SPLINE
SPL {X  -165.650, Y  +492.090, Z    +0.000, E1   -45.292, E3 +369321.420}
SPL {X  -165.650, Y  +498.857, Z    +0.000, E1   -45.339, E3 +369334.757}
SPL {X  -165.650, Y  +505.115, Z    +0.000, E1   -45.299, E3 +369347.706}
SPL {X  -165.650, Y  +510.931, Z    +0.000, E1   -45.250, E3 +369359.696}
SPL {X  -165.650, Y  +516.157, Z    +0.000, E1   -45.240, E3 +369370.371}
SPL {X  -165.650, Y  +521.049, Z    +0.000, E1   -45.236, E3 +369380.323}
SPL {X  -165.650, Y  +527.050, Z    +0.000, E1   -45.345, E3 +369391.820}
SPL {X  -165.650, Y  +532.042, Z    +0.000, E1   -45.233, E3 +369402.563}
SPL {X  -165.650, Y  +537.290, Z    +0.000, E1   -45.204, E3 +369413.404}
SPL {X  -165.650, Y  +544.196, Z    +0.000, E1   -45.432, E3 +369426.078}
SPL {X  -165.650, Y  +548.678, Z    +0.000, E1   -45.162, E3 +369436.642}
SPL {X  -165.650, Y  +554.600, Z    +0.000, E1   -45.345, E3 +369447.619}
SPL {X  -165.650, Y  +559.896, Z    +0.000, E1   -45.150, E3 +369459.474}
SPL {X  -165.650, Y  +566.830, Z    +0.000, E1   -45.346, E3 +369472.454}
SPL {X  -165.650, Y  +573.074, Z    +0.000, E1   -45.379, E3 +369484.785}
SPL {X  -165.650, Y  +579.360, Z    +0.000, E1   -45.300, E3 +369498.070}
SPL {X  -165.650, Y  +584.577, Z    +0.000, E1   -45.167, E3 +369509.293}
SPL {X  -165.650, Y  +590.060, Z    +0.000, E1   -45.221, E3 +369520.184}
SPL {X  -165.650, Y  +596.611, Z    +0.000, E1   -45.390, E3 +369532.421}
SPL {X  -165.650, Y  +603.637, Z    +0.000, E1   -45.296, E3 +369547.339}
SPL {X  -165.650, Y  +610.850, Z    +0.000, E1   -45.208, E3 +369562.348}
SPL {X  -165.650, Y  +617.450, Z    +0.000, E1   -45.402, E3 +369574.550}
SPL {X  -165.650, Y  +622.720, Z    +0.000, E1   -45.272, E3 +369585.948}
SPL {X  -165.650, Y  +627.828, Z    +0.000, E1   -45.174, E3 +369596.904}
SPL {X  -165.650, Y  +634.620, Z    +0.000, E1   -45.438, E3 +369609.110}
SPL {X  -165.650, Y  +640.808, Z    +0.000, E1   -45.294, E3 +369622.484}
SPL {X  -165.650, Y  +646.552, Z    +0.000, E1   -45.137, E3 +369635.009}
SPL {X  -165.650, Y  +652.431, Z    +0.000, E1   -45.333, E3 +369645.763}
SPL {X  -165.650, Y  +657.443, Z    +0.000, E1   -45.316, E3 +369656.020}
SPL {X  -165.650, Y  +662.999, Z    +0.000, E1   -45.214, E3 +369667.892}
SPL {X  -165.650, Y  +668.737, Z    +0.000, E1   -45.236, E3 +369679.406}
SPL {X  -165.650, Y  +675.226, Z    +0.000, E1   -45.503, E3 +369690.910}
SPL {X  -165.597, Y  +679.672, Z    +0.000, E1   -45.206, E3 +369701.631}
SPL {X  -165.388, Y  +684.808, Z    +0.000, E1   -45.192, E3 +369712.139}
SPL {X  -165.020, Y  +689.938, Z    +0.000, E1   -45.107, E3 +369723.082}
SPL {X  -164.358, Y  +696.147, Z    +0.000, E1   -45.160, E3 +369735.347}
SPL {X  -163.631, Y  +701.286, Z    +0.000, E1   -44.994, E3 +369746.639}
SPL {X  -162.679, Y  +706.734, Z    +0.000, E1   -44.812, E3 +369758.872}
SPL {X  -161.655, Y  +711.661, Z    +0.000, E1   -44.525, E3 +369770.253}
SPL {X  -160.692, Y  +715.726, Z    +0.000, E1   -44.379, E3 +369779.411}
SPL {X  -159.384, Y  +720.631, Z    +0.000, E1   -44.155, E3 +369790.561}
SPL {X  -158.321, Y  +724.227, Z    +0.000, E1   -43.955, E3 +369798.882}
SPL {X  -156.604, Y  +729.490, Z    +0.000, E1   -44.229, E3 +369808.049}
SPL {X  -147.100, Y  +751.668, Z    +0.000, E1   -50.624, E3 +369813.935}
SPL {X  -144.116, Y  +757.172, Z    +0.000, E1   -42.809, E3 +369883.332}
SPL {X  -127.227, Y  +781.582, Z    +0.000, E1   -46.780, E3 +369929.001}
ENDSPLINE

SPLINE
SPL {X  -133.736, Y  +773.248, Z    +0.000, E1   -45.385, E3 +370007.044}
SPL {X  -160.761, Y  +715.447, Z    +0.000, E1   -23.748, E3 +369963.893}
SPL {X  -164.304, Y  +696.571, Z    +0.000, E1   -14.525, E3 +369969.117}
SPL {X  -165.498, Y  +682.585, Z    +0.000, E1    -6.769, E3 +369968.792}
SPL {X  -165.650, Y  +674.975, Z    +0.000, E1    -1.888, E3 +369967.150}
SPL {X  -165.650, Y  +671.520, Z    +0.000, E1    +0.682, E3 +369966.077}
SPL {X  -165.650, Y  +668.289, Z    +0.000, E1    +3.417, E3 +369965.919}
SPL {X  -165.650, Y  +663.040, Z    +0.000, E1    +8.602, E3 +369965.114}
SPL {X  -165.650, Y  +655.692, Z    +0.000, E1   +17.061, E3 +369963.649}
SPL {X  -165.650, Y  +646.511, Z    +0.000, E1   +26.434, E3 +369966.429}
SPL {X  -165.650, Y  +637.905, Z    +0.000, E1   +40.225, E3 +369954.554}
SPL {X  -165.650, Y  +611.479, Z    +0.000, E1   +52.226, E3 +369968.106}
SPL {X  -165.650, Y  +599.923, Z    +0.000, E1   +51.240, E3 +369985.195}
SPL {X  -165.650, Y  +553.219, Z    +0.000, E1   +52.865, E3 +370041.956}
ENDSPLINE

SPLINE
SPL {X  -165.650, Y  +569.883, Z    +0.000, E1   +45.183, E3 +370057.633}
ENDSPLINE

SPLINE
SPL {X  -165.650, Y  +561.960, Z    +0.000, E1   +45.285, E3 +370073.288}
SPL {X  -165.650, Y  +554.065, Z    +0.000, E1   +45.254, E3 +370089.350}
SPL {X  -165.650, Y  +548.074, Z    +0.000, E1   +45.245, E3 +370101.461}
SPL {X  -165.650, Y  +542.958, Z    +0.000, E1   +45.131, E3 +370112.591}
SPL {X  -165.650, Y  +535.288, Z    +0.000, E1   +45.332, E3 +370127.032}
SPL {X  -165.650, Y  +529.160, Z    +0.000, E1   +45.215, E3 +370140.013}
SPL {X  -165.650, Y  +522.672, Z    +0.000, E1   +45.331, E3 +370152.579}
SPL {X  -165.650, Y  +516.211, Z    +0.000, E1   +45.175, E3 +370166.539}
SPL {X  -165.650, Y  +509.762, Z    +0.000, E1   +45.191, E3 +370179.581}
SPL {X  -165.650, Y  +503.812, Z    +0.000, E1   +45.188, E3 +370191.620}
SPL {X  -165.650, Y  +499.646, Z    +0.000, E1   +44.886, E3 +370201.891}
ENDSPLINE

SPLINE
SPL {X  -165.650, Y  +516.930, Z    +0.000, E1   +36.544, E3 +370210.561}
ENDSPLINE

SPLINE
SPL {X  -165.650, Y  +511.324, Z    +0.000, E1   +37.254, E3 +370221.552}
SPL {X  -165.650, Y  +504.742, Z    +0.000, E1   +38.087, E3 +370233.857}
SPL {X  -165.650, Y  +497.845, Z    +0.000, E1   +39.022, E3 +370245.932}
SPL {X  -165.650, Y  +491.819, Z    +0.000, E1   +39.756, E3 +370256.451}
SPL {X  -165.650, Y  +485.086, Z    +0.000, E1   +40.678, E3 +370267.295}
SPL {X  -165.650, Y  +476.633, Z    +0.000, E1   +41.847, E3 +370279.994}
SPL {X  -165.650, Y  +468.596, Z    +0.000, E1   +42.673, E3 +370293.257}
SPL {X  -165.650, Y  +460.562, Z    +0.000, E1   +43.733, E3 +370304.409}
SPL {X  -165.650, Y  +455.629, Z    +0.000, E1   +44.293, E3 +370311.528}
SPL {X  -165.650, Y  +449.099, Z    +0.000, E1   +44.871, E3 +370321.760}
SPL {X  -165.650, Y  +442.120, Z    +0.000, E1   +45.313, E3 +370333.312}
SPL {X  -165.650, Y  +439.103, Z    +0.000, E1   +44.726, E3 +370342.921}
SPL {X  -165.650, Y  +433.421, Z    +0.000, E1   +45.110, E3 +370352.309}
SPL {X  -165.650, Y  +426.476, Z    +0.000, E1   +45.244, E3 +370365.812}
SPL {X  -165.650, Y  +420.418, Z    +0.000, E1   +45.128, E3 +370378.606}
SPL {X  -165.650, Y  +415.564, Z    +0.000, E1   +45.195, E3 +370388.151}
SPL {X  -165.650, Y  +410.687, Z    +0.000, E1   +44.955, E3 +370399.467}
SPL {X  -165.650, Y  +402.778, Z    +0.000, E1   +45.323, E3 +370413.548}
SPL {X  -165.650, Y  +396.171, Z    +0.000, E1   +44.969, E3 +370428.969}
SPL {X  -165.650, Y  +390.060, Z    +0.000, E1   +45.007, E3 +370441.202}
SPL {X  -165.650, Y  +383.700, Z    +0.000, E1   +45.345, E3 +370452.126}
SPL {X  -165.650, Y  +379.225, Z    +0.000, E1   +45.073, E3 +370462.815}
SPL {X  -165.591, Y  +374.097, Z    +0.000, E1   +45.069, E3 +370473.296}
SPL {X  -165.372, Y  +368.914, Z    +0.000, E1   +45.103, E3 +370483.656}
SPL {X  -164.833, Y  +362.064, Z    +0.000, E1   +44.999, E3 +370498.441}
SPL {X  -164.024, Y  +355.348, Z    +0.000, E1   +45.002, E3 +370511.829}
SPL {X  -163.441, Y  +351.538, Z    +0.000, E1   +44.749, E3 +370521.045}
SPL {X  -162.419, Y  +345.942, Z    +0.000, E1   +44.540, E3 +370533.777}
SPL {X  -161.210, Y  +340.404, Z    +0.000, E1   +44.250, E3 +370546.602}
SPL {X  -159.961, Y  +335.460, Z    +0.000, E1   +44.205, E3 +370556.965}
SPL {X  -158.595, Y  +330.672, Z    +0.000, E1   +43.797, E3 +370568.943}
SPL {X  -156.695, Y  +324.773, Z    +0.000, E1   +43.987, E3 +370579.840}
SPL {X  -148.318, Y  +304.733, Z    +0.000, E1   +49.897, E3 +370585.076}
SPL {X  -138.435, Y  +287.529, Z    +0.000, E1   +45.834, E3 +370650.401}
SPL {X  -134.645, Y  +282.008, Z    +0.000, E1   +45.207, E3 +370680.057}
ENDSPLINE

SPLINE
SPL {X  -154.915, Y  +319.839, Z    +0.000, E1   +31.584, E3 +370739.576}
SPL {X  -161.387, Y  +341.161, Z    +0.000, E1   +22.590, E3 +370753.422}
SPL {X  -164.566, Y  +359.576, Z    +0.000, E1   +13.425, E3 +370732.015}
SPL {X  -165.355, Y  +368.611, Z    +0.000, E1    +8.407, E3 +370735.596}
SPL {X  -165.614, Y  +375.050, Z    +0.000, E1    +4.520, E3 +370736.900}
SPL {X  -165.650, Y  +379.847, Z    +0.000, E1    +1.364, E3 +370735.249}
SPL {X  -165.650, Y  +383.246, Z    +0.000, E1    -1.216, E3 +370734.343}
SPL {X  -165.650, Y  +386.866, Z    +0.000, E1    -4.337, E3 +370734.395}
SPL {X  -165.650, Y  +394.200, Z    +0.000, E1   -11.943, E3 +370732.162}
SPL {X  -165.650, Y  +405.401, Z    +0.000, E1   -24.512, E3 +370731.982}
SPL {X  -165.650, Y  +418.038, Z    +0.000, E1   -38.688, E3 +370728.210}
SPL {X  -165.650, Y  +461.620, Z    +0.000, E1   -55.594, E3 +370748.388}
SPL {X  -165.650, Y  +498.574, Z    +0.000, E1   -52.082, E3 +370809.414}
ENDSPLINE

SPLINE
SPL {X  -165.650, Y  +484.983, Z    +0.000, E1   -45.406, E3 +370824.916}
ENDSPLINE

SPLINE
SPL {X  -165.650, Y  +492.090, Z    +0.000, E1   -45.292, E3 +370839.939}
SPL {X  -165.650, Y  +498.857, Z    +0.000, E1   -45.339, E3 +370853.276}
SPL {X  -165.650, Y  +505.115, Z    +0.000, E1   -45.299, E3 +370866.224}
SPL {X  -165.650, Y  +510.931, Z    +0.000, E1   -45.250, E3 +370878.215}
SPL {X  -165.650, Y  +516.157, Z    +0.000, E1   -45.240, E3 +370888.889}
SPL {X  -165.650, Y  +521.049, Z    +0.000, E1   -45.236, E3 +370898.842}
SPL {X  -165.650, Y  +527.050, Z    +0.000, E1   -45.345, E3 +370910.338}
SPL {X  -165.650, Y  +532.042, Z    +0.000, E1   -45.233, E3 +370921.081}
SPL {X  -165.650, Y  +537.290, Z    +0.000, E1   -45.204, E3 +370931.922}
SPL {X  -165.650, Y  +544.196, Z    +0.000, E1   -45.432, E3 +370944.597}
SPL {X  -165.650, Y  +548.678, Z    +0.000, E1   -45.162, E3 +370955.160}
SPL {X  -165.650, Y  +554.600, Z    +0.000, E1   -45.345, E3 +370966.137}
SPL {X  -165.650, Y  +559.896, Z    +0.000, E1   -45.150, E3 +370977.993}
SPL {X  -165.650, Y  +566.830, Z    +0.000, E1   -45.346, E3 +370990.973}
SPL {X  -165.650, Y  +573.074, Z    +0.000, E1   -45.379, E3 +371003.304}
SPL {X  -165.650, Y  +579.360, Z    +0.000, E1   -45.300, E3 +371016.589}
SPL {X  -165.650, Y  +584.577, Z    +0.000, E1   -45.167, E3 +371027.812}
SPL {X  -165.650, Y  +590.060, Z    +0.000, E1   -45.221, E3 +371038.703}
SPL {X  -165.650, Y  +596.611, Z    +0.000, E1   -45.390, E3 +371050.939}
SPL {X  -165.650, Y  +603.637, Z    +0.000, E1   -45.296, E3 +371065.858}
SPL {X  -165.650, Y  +610.850, Z    +0.000, E1   -45.208, E3 +371080.866}
SPL {X  -165.650, Y  +617.450, Z    +0.000, E1   -45.402, E3 +371093.069}
SPL {X  -165.650, Y  +622.720, Z    +0.000, E1   -45.272, E3 +371104.466}
SPL {X  -165.650, Y  +627.828, Z    +0.000, E1   -45.174, E3 +371115.423}
SPL {X  -165.650, Y  +634.620, Z    +0.000, E1   -45.438, E3 +371127.629}
SPL {X  -165.650, Y  +640.808, Z    +0.000, E1   -45.294, E3 +371141.003}
SPL {X  -165.650, Y  +646.552, Z    +0.000, E1   -45.137, E3 +371153.527}
SPL {X  -165.650, Y  +652.431, Z    +0.000, E1   -45.333, E3 +371164.282}
SPL {X  -165.650, Y  +657.443, Z    +0.000, E1   -45.316, E3 +371174.538}
SPL {X  -165.650, Y  +662.999, Z    +0.000, E1   -45.214, E3 +371186.410}
SPL {X  -165.650, Y  +668.737, Z    +0.000, E1   -45.236, E3 +371197.925}
SPL {X  -165.650, Y  +675.226, Z    +0.000, E1   -45.503, E3 +371209.429}
SPL {X  -165.597, Y  +679.672, Z    +0.000, E1   -45.206, E3 +371220.150}
SPL {X  -165.388, Y  +684.808, Z    +0.000, E1   -45.192, E3 +371230.657}
SPL {X  -165.020, Y  +689.938, Z    +0.000, E1   -45.107, E3 +371241.600}
SPL {X  -164.358, Y  +696.147, Z    +0.000, E1   -45.160, E3 +371253.866}
SPL {X  -163.631, Y  +701.286, Z    +0.000, E1   -44.994, E3 +371265.158}
SPL {X  -162.679, Y  +706.734, Z    +0.000, E1   -44.812, E3 +371277.391}
SPL {X  -161.655, Y  +711.661, Z    +0.000, E1   -44.525, E3 +371288.772}
SPL {X  -160.692, Y  +715.726, Z    +0.000, E1   -44.379, E3 +371297.929}
SPL {X  -159.384, Y  +720.631, Z    +0.000, E1   -44.155, E3 +371309.079}
SPL {X  -158.321, Y  +724.227, Z    +0.000, E1   -43.955, E3 +371317.400}
SPL {X  -156.604, Y  +729.490, Z    +0.000, E1   -44.229, E3 +371326.567}
SPL {X  -147.100, Y  +751.668, Z    +0.000, E1   -50.624, E3 +371332.454}
SPL {X  -144.116, Y  +757.172, Z    +0.000, E1   -42.809, E3 +371401.850}
SPL {X  -127.227, Y  +781.582, Z    +0.000, E1   -46.780, E3 +371447.520}
ENDSPLINE

SPLINE
SPL {X  -133.736, Y  +773.248, Z    +0.000, E1   -45.385, E3 +371525.562}
SPL {X  -160.761, Y  +715.447, Z    +0.000, E1   -23.748, E3 +371482.412}
SPL {X  -164.304, Y  +696.571, Z    +0.000, E1   -14.525, E3 +371487.636}
SPL {X  -165.498, Y  +682.585, Z    +0.000, E1    -6.769, E3 +371487.310}
SPL {X  -165.650, Y  +674.975, Z    +0.000, E1    -1.888, E3 +371485.668}
SPL {X  -165.650, Y  +671.520, Z    +0.000, E1    +0.682, E3 +371484.596}
SPL {X  -165.650, Y  +668.289, Z    +0.000, E1    +3.417, E3 +371484.438}
SPL {X  -165.650, Y  +663.040, Z    +0.000, E1    +8.602, E3 +371483.632}
SPL {X  -165.650, Y  +655.692, Z    +0.000, E1   +17.061, E3 +371482.167}
SPL {X  -165.650, Y  +646.511, Z    +0.000, E1   +26.434, E3 +371484.948}
SPL {X  -165.650, Y  +637.905, Z    +0.000, E1   +40.225, E3 +371473.072}
SPL {X  -165.650, Y  +611.479, Z    +0.000, E1   +52.226, E3 +371486.625}
SPL {X  -165.650, Y  +599.923, Z    +0.000, E1   +51.240, E3 +371503.714}
SPL {X  -165.650, Y  +553.219, Z    +0.000, E1   +52.865, E3 +371560.474}
ENDSPLINE

SPLINE
SPL {X  -165.650, Y  +569.883, Z    +0.000, E1   +45.183, E3 +371576.151}
ENDSPLINE

SPLINE
SPL {X  -165.650, Y  +561.960, Z    +0.000, E1   +45.285, E3 +371591.807}
SPL {X  -165.650, Y  +554.065, Z    +0.000, E1   +45.254, E3 +371607.868}
SPL {X  -165.650, Y  +548.074, Z    +0.000, E1   +45.245, E3 +371619.979}
SPL {X  -165.650, Y  +542.958, Z    +0.000, E1   +45.131, E3 +371631.110}
SPL {X  -165.650, Y  +535.288, Z    +0.000, E1   +45.332, E3 +371645.551}
SPL {X  -165.650, Y  +529.160, Z    +0.000, E1   +45.215, E3 +371658.532}
SPL {X  -165.650, Y  +522.672, Z    +0.000, E1   +45.331, E3 +371671.098}
SPL {X  -165.650, Y  +516.211, Z    +0.000, E1   +45.175, E3 +371685.057}
SPL {X  -165.650, Y  +509.762, Z    +0.000, E1   +45.191, E3 +371698.099}
SPL {X  -165.650, Y  +503.812, Z    +0.000, E1   +45.188, E3 +371710.138}
SPL {X  -165.650, Y  +499.646, Z    +0.000, E1   +44.886, E3 +371720.409}
ENDSPLINE

SPLINE
SPL {X  -165.650, Y  +514.834, Z    +0.000, E1   +36.829, E3 +371733.175}
ENDSPLINE

SPLINE
SPL {X  -165.650, Y  +506.421, Z    +0.000, E1   +37.886, E3 +371749.287}
SPL {X  -165.650, Y  +499.917, Z    +0.000, E1   +38.752, E3 +371760.748}
SPL {X  -165.650, Y  +493.826, Z    +0.000, E1   +39.521, E3 +371771.502}
SPL {X  -165.650, Y  +487.003, Z    +0.000, E1   +40.380, E3 +371782.956}
SPL {X  -165.650, Y  +478.382, Z    +0.000, E1   +41.628, E3 +371795.869}
SPL {X  -165.650, Y  +472.112, Z    +0.000, E1   +42.202, E3 +371806.608}
SPL {X  -165.650, Y  +466.741, Z    +0.000, E1   +42.890, E3 +371814.529}
SPL {X  -165.650, Y  +458.202, Z    +0.000, E1   +44.020, E3 +371826.316}
SPL {X  -165.650, Y  +449.099, Z    +0.000, E1   +44.871, E3 +371840.279}
SPL {X  -165.650, Y  +442.120, Z    +0.000, E1   +45.313, E3 +371851.831}
SPL {X  -165.650, Y  +436.063, Z    +0.000, E1   +44.972, E3 +371866.415}
SPL {X  -165.650, Y  +427.943, Z    +0.000, E1   +45.362, E3 +371880.452}
SPL {X  -165.650, Y  +422.523, Z    +0.000, E1   +45.103, E3 +371893.131}
SPL {X  -165.650, Y  +415.564, Z    +0.000, E1   +45.195, E3 +371906.670}
SPL {X  -165.650, Y  +410.687, Z    +0.000, E1   +44.955, E3 +371917.986}
SPL {X  -165.650, Y  +405.522, Z    +0.000, E1   +45.119, E3 +371927.546}
SPL {X  -165.650, Y  +399.216, Z    +0.000, E1   +45.246, E3 +371939.740}
SPL {X  -165.650, Y  +391.618, Z    +0.000, E1   +45.037, E3 +371956.518}
SPL {X  -165.650, Y  +383.700, Z    +0.000, E1   +45.345, E3 +371970.644}
SPL {X  -165.650, Y  +379.225, Z    +0.000, E1   +45.073, E3 +371981.333}
SPL {X  -165.591, Y  +374.097, Z    +0.000, E1   +45.069, E3 +371991.814}
SPL {X  -165.372, Y  +368.914, Z    +0.000, E1   +45.103, E3 +372002.174}
SPL {X  -164.987, Y  +363.696, Z    +0.000, E1   +45.006, E3 +372013.397}
SPL {X  -164.256, Y  +357.053, Z    +0.000, E1   +44.969, E3 +372027.200}
SPL {X  -163.441, Y  +351.538, Z    +0.000, E1   +44.749, E3 +372039.564}
SPL {X  -162.419, Y  +345.942, Z    +0.000, E1   +44.540, E3 +372052.295}
SPL {X  -161.210, Y  +340.404, Z    +0.000, E1   +44.250, E3 +372065.120}
SPL {X  -159.961, Y  +335.460, Z    +0.000, E1   +44.205, E3 +372075.483}
SPL {X  -158.595, Y  +330.672, Z    +0.000, E1   +43.797, E3 +372087.461}
SPL {X  -156.695, Y  +324.773, Z    +0.000, E1   +43.987, E3 +372098.358}
SPL {X  -148.318, Y  +304.733, Z    +0.000, E1   +49.897, E3 +372103.595}
SPL {X  -138.435, Y  +287.529, Z    +0.000, E1   +45.834, E3 +372168.919}
SPL {X  -137.083, Y  +285.505, Z    +0.000, E1   +44.955, E3 +372187.084}
ENDSPLINE

SPLINE
SPL {X  -137.518, Y  +286.149, Z    +0.000, E1   +42.648, E3 +372250.964}
SPL {X  -156.430, Y  +324.005, Z    +0.000, E1   +29.926, E3 +372256.099}
SPL {X  -161.387, Y  +341.161, Z    +0.000, E1   +22.590, E3 +372271.940}
SPL {X  -164.566, Y  +359.576, Z    +0.000, E1   +13.425, E3 +372250.534}
SPL {X  -165.355, Y  +368.611, Z    +0.000, E1    +8.407, E3 +372254.115}
SPL {X  -165.614, Y  +375.050, Z    +0.000, E1    +4.520, E3 +372255.418}
SPL {X  -165.650, Y  +379.847, Z    +0.000, E1    +1.364, E3 +372253.768}
SPL {X  -165.650, Y  +383.246, Z    +0.000, E1    -1.216, E3 +372252.861}
SPL {X  -165.650, Y  +386.866, Z    +0.000, E1    -4.337, E3 +372252.914}
SPL {X  -165.650, Y  +394.200, Z    +0.000, E1   -11.943, E3 +372250.681}
SPL {X  -165.650, Y  +405.401, Z    +0.000, E1   -24.512, E3 +372250.501}
SPL {X  -165.650, Y  +418.038, Z    +0.000, E1   -38.688, E3 +372246.728}
SPL {X  -165.650, Y  +461.620, Z    +0.000, E1   -55.594, E3 +372266.907}
SPL {X  -165.650, Y  +498.574, Z    +0.000, E1   -52.082, E3 +372327.932}
ENDSPLINE

SPLINE
SPL {X  -165.650, Y  +484.983, Z    +0.000, E1   -45.406, E3 +372343.435}
ENDSPLINE

SPLINE
SPL {X  -165.650, Y  +492.090, Z    +0.000, E1   -45.292, E3 +372358.457}
SPL {X  -165.650, Y  +498.857, Z    +0.000, E1   -45.339, E3 +372371.794}
SPL {X  -165.650, Y  +505.115, Z    +0.000, E1   -45.299, E3 +372384.743}
SPL {X  -165.650, Y  +510.931, Z    +0.000, E1   -45.250, E3 +372396.734}
SPL {X  -165.650, Y  +516.157, Z    +0.000, E1   -45.240, E3 +372407.408}
SPL {X  -165.650, Y  +521.049, Z    +0.000, E1   -45.236, E3 +372417.360}
SPL {X  -165.650, Y  +527.050, Z    +0.000, E1   -45.345, E3 +372428.857}
SPL {X  -165.650, Y  +532.042, Z    +0.000, E1   -45.233, E3 +372439.600}
SPL {X  -165.650, Y  +537.290, Z    +0.000, E1   -45.204, E3 +372450.441}
SPL {X  -165.650, Y  +544.196, Z    +0.000, E1   -45.432, E3 +372463.115}
SPL {X  -165.650, Y  +548.678, Z    +0.000, E1   -45.162, E3 +372473.679}
SPL {X  -165.650, Y  +554.600, Z    +0.000, E1   -45.345, E3 +372484.656}
SPL {X  -165.650, Y  +559.896, Z    +0.000, E1   -45.150, E3 +372496.511}
SPL {X  -165.650, Y  +566.830, Z    +0.000, E1   -45.346, E3 +372509.491}
SPL {X  -165.650, Y  +573.074, Z    +0.000, E1   -45.379, E3 +372521.822}
SPL {X  -165.650, Y  +579.360, Z    +0.000, E1   -45.300, E3 +372535.107}
SPL {X  -165.650, Y  +584.577, Z    +0.000, E1   -45.167, E3 +372546.330}
SPL {X  -165.650, Y  +590.060, Z    +0.000, E1   -45.221, E3 +372557.221}
SPL {X  -165.650, Y  +596.611, Z    +0.000, E1   -45.390, E3 +372569.458}
SPL {X  -165.650, Y  +601.960, Z    +0.000, E1   -45.255, E3 +372581.066}
SPL {X  -165.650, Y  +605.976, Z    +0.000, E1   -45.260, E3 +372589.116}
SPL {X  -165.650, Y  +610.850, Z    +0.000, E1   -45.208, E3 +372599.385}
SPL {X  -165.650, Y  +617.450, Z    +0.000, E1   -45.402, E3 +372611.587}
SPL {X  -165.650, Y  +622.720, Z    +0.000, E1   -45.272, E3 +372622.985}
SPL {X  -165.650, Y  +627.828, Z    +0.000, E1   -45.174, E3 +372633.941}
SPL {X  -165.650, Y  +634.620, Z    +0.000, E1   -45.438, E3 +372646.147}
SPL {X  -165.650, Y  +640.808, Z    +0.000, E1   -45.294, E3 +372659.521}
SPL {X  -165.650, Y  +646.552, Z    +0.000, E1   -45.137, E3 +372672.046}
SPL {X  -165.650, Y  +652.431, Z    +0.000, E1   -45.333, E3 +372682.800}
SPL {X  -165.650, Y  +657.443, Z    +0.000, E1   -45.316, E3 +372693.057}
SPL {X  -165.650, Y  +662.999, Z    +0.000, E1   -45.214, E3 +372704.929}
SPL {X  -165.650, Y  +668.737, Z    +0.000, E1   -45.236, E3 +372716.443}
SPL {X  -165.650, Y  +675.226, Z    +0.000, E1   -45.503, E3 +372727.947}
SPL {X  -165.597, Y  +679.672, Z    +0.000, E1   -45.206, E3 +372738.668}
SPL {X  -165.388, Y  +684.808, Z    +0.000, E1   -45.192, E3 +372749.176}
SPL {X  -165.020, Y  +689.938, Z    +0.000, E1   -45.107, E3 +372760.119}
SPL {X  -164.358, Y  +696.147, Z    +0.000, E1   -45.160, E3 +372772.384}
SPL {X  -163.631, Y  +701.286, Z    +0.000, E1   -44.994, E3 +372783.676}
SPL {X  -163.047, Y  +704.748, Z    +0.000, E1   -44.682, E3 +372792.500}
SPL {X  -161.884, Y  +710.619, Z    +0.000, E1   -44.738, E3 +372804.125}
SPL {X  -160.692, Y  +715.726, Z    +0.000, E1   -44.379, E3 +372816.448}
SPL {X  -159.384, Y  +720.631, Z    +0.000, E1   -44.155, E3 +372827.598}
SPL {X  -157.745, Y  +726.062, Z    +0.000, E1   -43.902, E3 +372840.084}
SPL {X  -153.030, Y  +738.918, Z    +0.000, E1   -47.123, E3 +372847.687}
SPL {X  -145.149, Y  +755.323, Z    +0.000, E1   -51.167, E3 +372853.819}
SPL {X  -143.038, Y  +759.047, Z    +0.000, E1   -43.157, E3 +372922.992}
SPL {X  -123.277, Y  +786.146, Z    +0.000, E1   -47.533, E3 +372979.048}
ENDSPLINE

SPLINE
SPL {X  -133.736, Y  +773.248, Z    +0.000, E1   -45.385, E3 +373044.081}
SPL {X  -160.761, Y  +715.447, Z    +0.000, E1   -23.748, E3 +373000.930}
SPL {X  -164.304, Y  +696.571, Z    +0.000, E1   -14.525, E3 +373006.154}
SPL {X  -165.498, Y  +682.585, Z    +0.000, E1    -6.769, E3 +373005.829}
SPL {X  -165.650, Y  +674.975, Z    +0.000, E1    -1.888, E3 +373004.187}
SPL {X  -165.650, Y  +670.481, Z    +0.000, E1    +1.454, E3 +373003.628}
SPL {X  -165.650, Y  +665.304, Z    +0.000, E1    +6.303, E3 +373002.131}
SPL {X  -165.650, Y  +657.587, Z    +0.000, E1   +14.733, E3 +373000.905}
SPL {X  -165.650, Y  +646.511, Z    +0.000, E1   +26.434, E3 +373003.466}
SPL {X  -165.650, Y  +637.905, Z    +0.000, E1   +40.225, E3 +372991.591}
SPL {X  -165.650, Y  +611.479, Z    +0.000, E1   +52.226, E3 +373005.143}
SPL {X  -165.650, Y  +599.923, Z    +0.000, E1   +51.240, E3 +373022.232}
SPL {X  -165.650, Y  +553.219, Z    +0.000, E1   +52.865, E3 +373078.993}
ENDSPLINE

SPLINE
SPL {X  -165.650, Y  +569.883, Z    +0.000, E1   +45.183, E3 +373094.670}
ENDSPLINE

SPLINE
SPL {X  -165.650, Y  +561.960, Z    +0.000, E1   +45.285, E3 +373110.325}
SPL {X  -165.650, Y  +554.065, Z    +0.000, E1   +45.254, E3 +373126.387}
SPL {X  -165.650, Y  +548.074, Z    +0.000, E1   +45.245, E3 +373138.498}
SPL {X  -165.650, Y  +542.958, Z    +0.000, E1   +45.131, E3 +373149.628}
SPL {X  -165.650, Y  +535.288, Z    +0.000, E1   +45.332, E3 +373164.069}
SPL {X  -165.650, Y  +529.160, Z    +0.000, E1   +45.215, E3 +373177.050}
SPL {X  -165.650, Y  +522.672, Z    +0.000, E1   +45.331, E3 +373189.616}
SPL {X  -165.650, Y  +516.211, Z    +0.000, E1   +45.175, E3 +373203.576}
SPL {X  -165.650, Y  +509.762, Z    +0.000, E1   +45.191, E3 +373216.618}
SPL {X  -165.650, Y  +503.812, Z    +0.000, E1   +45.188, E3 +373228.657}
SPL {X  -165.650, Y  +499.646, Z    +0.000, E1   +44.886, E3 +373238.928}
ENDSPLINE

SPLINE
SPL {X  -165.650, Y  +514.834, Z    +0.000, E1   +36.829, E3 +373251.694}
ENDSPLINE

SPLINE
SPL {X  -165.650, Y  +506.421, Z    +0.000, E1   +37.886, E3 +373267.806}
SPL {X  -165.650, Y  +497.845, Z    +0.000, E1   +39.022, E3 +373282.969}
SPL {X  -165.650, Y  +488.971, Z    +0.000, E1   +40.149, E3 +373298.190}
SPL {X  -165.650, Y  +478.382, Z    +0.000, E1   +41.628, E3 +373314.387}
SPL {X  -165.650, Y  +468.596, Z    +0.000, E1   +42.673, E3 +373330.294}
SPL {X  -165.650, Y  +458.202, Z    +0.000, E1   +44.020, E3 +373344.835}
SPL {X  -165.650, Y  +449.761, Z    +0.000, E1   +45.086, E3 +373356.028}
SPL {X  -165.650, Y  +444.380, Z    +0.000, E1   +45.056, E3 +373367.347}
SPL {X  -165.650, Y  +436.063, Z    +0.000, E1   +44.972, E3 +373384.933}
SPL {X  -165.650, Y  +427.943, Z    +0.000, E1   +45.362, E3 +373398.971}
SPL {X  -165.650, Y  +422.523, Z    +0.000, E1   +45.103, E3 +373411.649}
SPL {X  -165.650, Y  +415.564, Z    +0.000, E1   +45.195, E3 +373425.188}
SPL {X  -165.650, Y  +410.687, Z    +0.000, E1   +44.955, E3 +373436.504}
SPL {X  -165.650, Y  +405.522, Z    +0.000, E1   +45.119, E3 +373446.064}
SPL {X  -165.650, Y  +399.216, Z    +0.000, E1   +45.246, E3 +373458.258}
SPL {X  -165.650, Y  +391.618, Z    +0.000, E1   +45.037, E3 +373475.036}
SPL {X  -165.650, Y  +383.700, Z    +0.000, E1   +45.345, E3 +373489.163}
SPL {X  -165.650, Y  +379.225, Z    +0.000, E1   +45.073, E3 +373499.852}
SPL {X  -165.591, Y  +374.097, Z    +0.000, E1   +45.069, E3 +373510.333}
SPL {X  -165.372, Y  +368.914, Z    +0.000, E1   +45.103, E3 +373520.693}
SPL {X  -164.833, Y  +362.064, Z    +0.000, E1   +44.999, E3 +373535.478}
SPL {X  -164.024, Y  +355.348, Z    +0.000, E1   +45.002, E3 +373548.866}
SPL {X  -163.140, Y  +349.774, Z    +0.000, E1   +44.687, E3 +373562.253}
SPL {X  -162.065, Y  +344.224, Z    +0.000, E1   +44.509, E3 +373574.342}
SPL {X  -161.210, Y  +340.404, Z    +0.000, E1   +44.250, E3 +373583.639}
SPL {X  -159.961, Y  +335.460, Z    +0.000, E1   +44.205, E3 +373594.002}
SPL {X  -158.595, Y  +330.672, Z    +0.000, E1   +43.797, E3 +373605.980}
SPL {X  -157.207, Y  +326.289, Z    +0.000, E1   +43.631, E3 +373615.733}
SPL {X  -152.192, Y  +313.097, Z    +0.000, E1   +47.715, E3 +373619.287}
SPL {X  -146.385, Y  +300.967, Z    +0.000, E1   +50.402, E3 +373625.482}
SPL {X  -138.435, Y  +287.529, Z    +0.000, E1   +45.834, E3 +373687.438}
SPL {X  -134.645, Y  +282.008, Z    +0.000, E1   +45.207, E3 +373717.094}
ENDSPLINE

SPLINE
SPL {X  -154.915, Y  +319.839, Z    +0.000, E1   +31.584, E3 +373776.613}
SPL {X  -161.387, Y  +341.161, Z    +0.000, E1   +22.590, E3 +373790.459}
SPL {X  -164.566, Y  +359.576, Z    +0.000, E1   +13.425, E3 +373769.052}
SPL {X  -165.355, Y  +368.611, Z    +0.000, E1    +8.407, E3 +373772.633}
SPL {X  -165.614, Y  +375.050, Z    +0.000, E1    +4.520, E3 +373773.937}
SPL {X  -165.650, Y  +379.271, Z    +0.000, E1    +1.752, E3 +373770.958}
SPL {X  -165.650, Y  +382.603, Z    +0.000, E1    -0.657, E3 +373772.166}
SPL {X  -165.650, Y  +386.866, Z    +0.000, E1    -4.337, E3 +373771.432}
SPL {X  -165.650, Y  +392.464, Z    +0.000, E1   -10.170, E3 +373769.436}
SPL {X  -165.650, Y  +397.361, Z    +0.000, E1   -15.736, E3 +373768.767}
SPL {X  -165.650, Y  +404.553, Z    +0.000, E1   -23.488, E3 +373769.544}
SPL {X  -165.650, Y  +415.773, Z    +0.000, E1   -36.308, E3 +373765.696}
SPL {X  -165.650, Y  +461.620, Z    +0.000, E1   -55.594, E3 +373785.425}
SPL {X  -165.650, Y  +505.847, Z    +0.000, E1   -55.467, E3 +373837.398}
ENDSPLINE

SPLINE
SPL {X  -165.650, Y  +495.538, Z    +0.000, E1   -50.621, E3 +373849.882}
SPL {X  -165.650, Y  +483.168, Z    +0.000, E1   -45.573, E3 +373857.107}
ENDSPLINE

SPLINE
SPL {X  -165.650, Y  +487.615, Z    +0.000, E1   -45.254, E3 +373868.129}
SPL {X  -165.650, Y  +493.602, Z    +0.000, E1   -45.283, E3 +373879.969}
SPL {X  -165.650, Y  +498.857, Z    +0.000, E1   -45.339, E3 +373890.313}
SPL {X  -165.650, Y  +504.159, Z    +0.000, E1   -45.384, E3 +373900.708}
SPL {X  -165.650, Y  +509.628, Z    +0.000, E1   -45.217, E3 +373912.891}
SPL {X  -165.650, Y  +516.157, Z    +0.000, E1   -45.240, E3 +373925.926}
SPL {X  -165.650, Y  +521.049, Z    +0.000, E1   -45.236, E3 +373935.879}
SPL {X  -165.650, Y  +527.050, Z    +0.000, E1   -45.345, E3 +373947.375}
SPL {X  -165.650, Y  +532.042, Z    +0.000, E1   -45.233, E3 +373958.118}
SPL {X  -165.650, Y  +537.290, Z    +0.000, E1   -45.204, E3 +373968.959}
SPL {X  -165.650, Y  +544.196, Z    +0.000, E1   -45.432, E3 +373981.634}
SPL {X  -165.650, Y  +548.678, Z    +0.000, E1   -45.162, E3 +373992.197}
SPL {X  -165.650, Y  +554.600, Z    +0.000, E1   -45.345, E3 +374003.174}
SPL {X  -165.650, Y  +559.896, Z    +0.000, E1   -45.150, E3 +374015.030}
SPL {X  -165.650, Y  +566.830, Z    +0.000, E1   -45.346, E3 +374028.010}
SPL {X  -165.650, Y  +573.074, Z    +0.000, E1   -45.379, E3 +374040.341}
SPL {X  -165.650, Y  +577.292, Z    +0.000, E1   -45.246, E3 +374049.604}
SPL {X  -165.650, Y  +583.131, Z    +0.000, E1   -45.255, E3 +374061.546}
SPL {X  -165.650, Y  +590.060, Z    +0.000, E1   -45.221, E3 +374075.740}
SPL {X  -165.650, Y  +596.611, Z    +0.000, E1   -45.390, E3 +374087.976}
SPL {X  -165.650, Y  +603.637, Z    +0.000, E1   -45.296, E3 +374102.895}
SPL {X  -165.650, Y  +610.850, Z    +0.000, E1   -45.208, E3 +374117.903}
SPL {X  -165.650, Y  +617.450, Z    +0.000, E1   -45.402, E3 +374130.106}
SPL {X  -165.650, Y  +622.720, Z    +0.000, E1   -45.272, E3 +374141.503}
SPL {X  -165.650, Y  +627.828, Z    +0.000, E1   -45.174, E3 +374152.460}
SPL {X  -165.650, Y  +636.061, Z    +0.000, E1   -45.380, E3 +374168.122}
SPL {X  -165.650, Y  +645.149, Z    +0.000, E1   -45.285, E3 +374187.053}
SPL {X  -165.650, Y  +652.431, Z    +0.000, E1   -45.333, E3 +374201.319}
SPL {X  -165.650, Y  +657.443, Z    +0.000, E1   -45.316, E3 +374211.575}
SPL {X  -165.650, Y  +662.999, Z    +0.000, E1   -45.214, E3 +374223.447}
SPL {X  -165.650, Y  +668.737, Z    +0.000, E1   -45.236, E3 +374234.962}
SPL {X  -165.650, Y  +675.226, Z    +0.000, E1   -45.503, E3 +374246.466}
SPL {X  -165.597, Y  +679.672, Z    +0.000, E1   -45.206, E3 +374257.187}
SPL {X  -165.388, Y  +684.808, Z    +0.000, E1   -45.192, E3 +374267.694}
SPL {X  -165.020, Y  +689.938, Z    +0.000, E1   -45.107, E3 +374278.637}
SPL {X  -164.358, Y  +696.147, Z    +0.000, E1   -45.160, E3 +374290.903}
SPL {X  -163.631, Y  +701.286, Z    +0.000, E1   -44.994, E3 +374302.195}
SPL {X  -163.047, Y  +704.748, Z    +0.000, E1   -44.682, E3 +374311.019}
SPL {X  -161.884, Y  +710.619, Z    +0.000, E1   -44.738, E3 +374322.644}
SPL {X  -160.692, Y  +715.726, Z    +0.000, E1   -44.379, E3 +374334.966}
SPL {X  -158.938, Y  +722.175, Z    +0.000, E1   -44.121, E3 +374349.614}
SPL {X  -156.604, Y  +729.490, Z    +0.000, E1   -44.229, E3 +374363.604}
SPL {X  -147.100, Y  +751.668, Z    +0.000, E1   -50.624, E3 +374369.491}
SPL {X  -143.038, Y  +759.047, Z    +0.000, E1   -43.157, E3 +374441.511}
SPL {X  -123.277, Y  +786.146, Z    +0.000, E1   -47.533, E3 +374497.566}
ENDSPLINE

SPLINE
SPL {X  -133.736, Y  +773.248, Z    +0.000, E1   -45.385, E3 +374562.599}
SPL {X  -160.761, Y  +715.447, Z    +0.000, E1   -23.748, E3 +374519.449}
SPL {X  -164.304, Y  +696.571, Z    +0.000, E1   -14.525, E3 +374524.673}
SPL {X  -165.374, Y  +685.052, Z    +0.000, E1    -8.166, E3 +374524.066}
SPL {X  -165.648, Y  +676.230, Z    +0.000, E1    -2.814, E3 +374523.217}
SPL {X  -165.650, Y  +670.481, Z    +0.000, E1    +1.454, E3 +374522.147}
SPL {X  -165.650, Y  +665.304, Z    +0.000, E1    +6.303, E3 +374520.649}
SPL {X  -165.650, Y  +657.587, Z    +0.000, E1   +14.733, E3 +374519.424}
SPL {X  -165.650, Y  +646.511, Z    +0.000, E1   +26.434, E3 +374521.985}
SPL {X  -165.650, Y  +637.905, Z    +0.000, E1   +40.225, E3 +374510.109}
SPL {X  -165.650, Y  +607.385, Z    +0.000, E1   +51.775, E3 +374529.867}
SPL {X  -165.650, Y  +598.058, Z    +0.000, E1   +51.157, E3 +374543.329}
SPL {X  -165.650, Y  +553.656, Z    +0.000, E1   +53.998, E3 +374590.328}
SPL {X  -165.650, Y  +553.154, Z    +0.000, E1   +52.102, E3 +374601.855}
ENDSPLINE

SPLINE
SPL {X  -165.650, Y  +569.883, Z    +0.000, E1   +45.183, E3 +374613.188}
ENDSPLINE

SPLINE
SPL {X  -165.650, Y  +564.081, Z    +0.000, E1   +45.208, E3 +374624.806}
SPL {X  -165.650, Y  +557.350, Z    +0.000, E1   +45.265, E3 +374638.243}
SPL {X  -165.650, Y  +549.414, Z    +0.000, E1   +45.294, E3 +374654.145}
SPL {X  -165.650, Y  +542.958, Z    +0.000, E1   +45.131, E3 +374668.147}
SPL {X  -165.650, Y  +535.288, Z    +0.000, E1   +45.332, E3 +374682.588}
SPL {X  -165.650, Y  +528.026, Z    +0.000, E1   +45.173, E3 +374698.246}
SPL {X  -165.650, Y  +520.964, Z    +0.000, E1   +45.458, E3 +374710.751}
SPL {X  -165.650, Y  +516.211, Z    +0.000, E1   +45.175, E3 +374722.094}
SPL {X  -165.650, Y  +511.047, Z    +0.000, E1   +45.193, E3 +374732.413}
SPL {X  -165.650, Y  +505.100, Z    +0.000, E1   +45.197, E3 +374744.616}
SPL {X  -165.650, Y  +499.646, Z    +0.000, E1   +44.886, E3 +374757.446}
ENDSPLINE

SPLINE
SPL {X  -165.650, Y  +516.930, Z    +0.000, E1   +36.544, E3 +374766.117}
ENDSPLINE

SPLINE
SPL {X  -165.650, Y  +511.324, Z    +0.000, E1   +37.254, E3 +374777.108}
SPL {X  -165.650, Y  +502.734, Z    +0.000, E1   +38.389, E3 +374792.876}
SPL {X  -165.650, Y  +493.826, Z    +0.000, E1   +39.521, E3 +374808.539}
SPL {X  -165.650, Y  +485.086, Z    +0.000, E1   +40.678, E3 +374822.851}
SPL {X  -165.650, Y  +476.633, Z    +0.000, E1   +41.847, E3 +374835.550}
SPL {X  -165.650, Y  +468.596, Z    +0.000, E1   +42.673, E3 +374848.812}
SPL {X  -165.650, Y  +460.562, Z    +0.000, E1   +43.733, E3 +374859.965}
SPL {X  -165.650, Y  +455.629, Z    +0.000, E1   +44.293, E3 +374867.084}
SPL {X  -165.650, Y  +449.099, Z    +0.000, E1   +44.871, E3 +374877.316}
SPL {X  -165.650, Y  +442.120, Z    +0.000, E1   +45.313, E3 +374888.868}
SPL {X  -165.650, Y  +436.063, Z    +0.000, E1   +44.972, E3 +374903.452}
SPL {X  -165.650, Y  +427.943, Z    +0.000, E1   +45.362, E3 +374917.489}
SPL {X  -165.650, Y  +422.523, Z    +0.000, E1   +45.103, E3 +374930.168}
SPL {X  -165.650, Y  +415.564, Z    +0.000, E1   +45.195, E3 +374943.707}
SPL {X  -165.650, Y  +410.687, Z    +0.000, E1   +44.955, E3 +374955.023}
SPL {X  -165.650, Y  +405.522, Z    +0.000, E1   +45.119, E3 +374964.583}
SPL {X  -165.650, Y  +399.216, Z    +0.000, E1   +45.246, E3 +374976.777}
SPL {X  -165.650, Y  +391.618, Z    +0.000, E1   +45.037, E3 +374993.555}
SPL {X  -165.650, Y  +383.700, Z    +0.000, E1   +45.345, E3 +375007.681}
SPL {X  -165.650, Y  +379.225, Z    +0.000, E1   +45.073, E3 +375018.370}
SPL {X  -165.591, Y  +374.097, Z    +0.000, E1   +45.069, E3 +375028.851}
SPL {X  -165.372, Y  +368.914, Z    +0.000, E1   +45.103, E3 +375039.211}
SPL {X  -164.987, Y  +363.696, Z    +0.000, E1   +45.006, E3 +375050.434}
SPL {X  -164.256, Y  +357.053, Z    +0.000, E1   +44.969, E3 +375064.237}
SPL {X  -163.441, Y  +351.538, Z    +0.000, E1   +44.749, E3 +375076.601}
SPL {X  -162.419, Y  +345.942, Z    +0.000, E1   +44.540, E3 +375089.332}
SPL {X  -161.210, Y  +340.404, Z    +0.000, E1   +44.250, E3 +375102.157}
SPL {X  -159.961, Y  +335.460, Z    +0.000, E1   +44.205, E3 +375112.520}
SPL {X  -158.595, Y  +330.672, Z    +0.000, E1   +43.797, E3 +375124.498}
SPL {X  -156.695, Y  +324.773, Z    +0.000, E1   +43.987, E3 +375135.395}
SPL {X  -148.318, Y  +304.733, Z    +0.000, E1   +49.897, E3 +375140.632}
SPL {X  -138.435, Y  +287.529, Z    +0.000, E1   +45.834, E3 +375205.956}
SPL {X  -134.645, Y  +282.008, Z    +0.000, E1   +45.207, E3 +375235.613}
ENDSPLINE

SPLINE
SPL {X  -154.915, Y  +319.839, Z    +0.000, E1   +31.584, E3 +375295.132}
SPL {X  -161.387, Y  +341.161, Z    +0.000, E1   +22.590, E3 +375308.977}
SPL {X  -164.566, Y  +359.576, Z    +0.000, E1   +13.425, E3 +375287.571}
SPL {X  -165.355, Y  +368.611, Z    +0.000, E1    +8.407, E3 +375291.152}
SPL {X  -165.614, Y  +375.050, Z    +0.000, E1    +4.520, E3 +375292.455}
SPL {X  -165.650, Y  +379.847, Z    +0.000, E1    +1.364, E3 +375290.805}
SPL {X  -165.650, Y  +383.246, Z    +0.000, E1    -1.216, E3 +375289.898}
SPL {X  -165.650, Y  +386.866, Z    +0.000, E1    -4.337, E3 +375289.951}
SPL {X  -165.650, Y  +394.200, Z    +0.000, E1   -11.943, E3 +375287.718}
SPL {X  -165.650, Y  +405.401, Z    +0.000, E1   -24.512, E3 +375287.538}
SPL {X  -165.650, Y  +418.038, Z    +0.000, E1   -38.688, E3 +375283.765}
SPL {X  -165.650, Y  +461.620, Z    +0.000, E1   -55.594, E3 +375303.944}
SPL {X  -165.650, Y  +498.574, Z    +0.000, E1   -52.082, E3 +375364.969}
ENDSPLINE

SPLINE
SPL {X  -165.650, Y  +483.168, Z    +0.000, E1   -45.573, E3 +375375.626}
ENDSPLINE

SPLINE
SPL {X  -165.650, Y  +487.615, Z    +0.000, E1   -45.254, E3 +375386.648}
SPL {X  -165.650, Y  +493.602, Z    +0.000, E1   -45.283, E3 +375398.488}
SPL {X  -165.650, Y  +498.857, Z    +0.000, E1   -45.339, E3 +375408.832}
SPL {X  -165.650, Y  +504.159, Z    +0.000, E1   -45.384, E3 +375419.226}
SPL {X  -165.650, Y  +509.628, Z    +0.000, E1   -45.217, E3 +375431.409}
SPL {X  -165.650, Y  +516.157, Z    +0.000, E1   -45.240, E3 +375444.445}
SPL {X  -165.650, Y  +521.049, Z    +0.000, E1   -45.236, E3 +375454.398}
SPL {X  -165.650, Y  +527.050, Z    +0.000, E1   -45.345, E3 +375465.894}
SPL {X  -165.650, Y  +532.042, Z    +0.000, E1   -45.233, E3 +375476.637}
SPL {X  -165.650, Y  +537.290, Z    +0.000, E1   -45.204, E3 +375487.478}
SPL {X  -165.650, Y  +544.196, Z    +0.000, E1   -45.432, E3 +375500.152}
SPL {X  -165.650, Y  +548.678, Z    +0.000, E1   -45.162, E3 +375510.716}
SPL {X  -165.650, Y  +554.600, Z    +0.000, E1   -45.345, E3 +375521.693}
SPL {X  -165.650, Y  +559.896, Z    +0.000, E1   -45.150, E3 +375533.548}
SPL {X  -165.650, Y  +566.830, Z    +0.000, E1   -45.346, E3 +375546.529}
SPL {X  -165.650, Y  +575.003, Z    +0.000, E1   -45.370, E3 +375563.013}
SPL {X  -165.650, Y  +583.131, Z    +0.000, E1   -45.255, E3 +375580.065}
SPL {X  -165.650, Y  +590.060, Z    +0.000, E1   -45.221, E3 +375594.258}
SPL {X  -165.650, Y  +596.611, Z    +0.000, E1   -45.390, E3 +375606.495}
SPL {X  -165.650, Y  +603.637, Z    +0.000, E1   -45.296, E3 +375621.414}
SPL {X  -165.650, Y  +610.850, Z    +0.000, E1   -45.208, E3 +375636.422}
SPL {X  -165.650, Y  +617.450, Z    +0.000, E1   -45.402, E3 +375648.624}
SPL {X  -165.650, Y  +622.720, Z    +0.000, E1   -45.272, E3 +375660.022}
SPL {X  -165.650, Y  +627.828, Z    +0.000, E1   -45.174, E3 +375670.978}
SPL {X  -165.650, Y  +636.061, Z    +0.000, E1   -45.380, E3 +375686.641}
SPL {X  -165.650, Y  +645.149, Z    +0.000, E1   -45.285, E3 +375705.571}
SPL {X  -165.650, Y  +652.431, Z    +0.000, E1   -45.333, E3 +375719.837}
SPL {X  -165.650, Y  +657.443, Z    +0.000, E1   -45.316, E3 +375730.094}
SPL {X  -165.650, Y  +662.999, Z    +0.000, E1   -45.214, E3 +375741.966}
SPL {X  -165.650, Y  +668.737, Z    +0.000, E1   -45.236, E3 +375753.481}
SPL {X  -165.650, Y  +675.226, Z    +0.000, E1   -45.503, E3 +375764.984}
SPL {X  -165.597, Y  +679.672, Z    +0.000, E1   -45.206, E3 +375775.705}
SPL {X  -165.388, Y  +684.808, Z    +0.000, E1   -45.192, E3 +375786.213}
SPL {X  -165.020, Y  +689.938, Z    +0.000, E1   -45.107, E3 +375797.156}
SPL {X  -164.358, Y  +696.147, Z    +0.000, E1   -45.160, E3 +375809.421}
SPL {X  -163.631, Y  +701.286, Z    +0.000, E1   -44.994, E3 +375820.713}
SPL {X  -163.047, Y  +704.748, Z    +0.000, E1   -44.682, E3 +375829.537}
SPL {X  -161.884, Y  +710.619, Z    +0.000, E1   -44.738, E3 +375841.162}
SPL {X  -160.692, Y  +715.726, Z    +0.000, E1   -44.379, E3 +375853.485}
SPL {X  -159.384, Y  +720.631, Z    +0.000, E1   -44.155, E3 +375864.635}
SPL {X  -158.321, Y  +724.227, Z    +0.000, E1   -43.955, E3 +375872.956}
SPL {X  -156.604, Y  +729.490, Z    +0.000, E1   -44.229, E3 +375882.123}
SPL {X  -147.100, Y  +751.668, Z    +0.000, E1   -50.624, E3 +375888.009}
SPL {X  -143.038, Y  +759.047, Z    +0.000, E1   -43.157, E3 +375960.029}
SPL {X  -123.277, Y  +786.146, Z    +0.000, E1   -47.533, E3 +376016.085}
ENDSPLINE

SPLINE
SPL {X  -133.736, Y  +773.248, Z    +0.000, E1   -45.385, E3 +376081.118}
SPL {X  -160.761, Y  +715.447, Z    +0.000, E1   -23.748, E3 +376037.967}
SPL {X  -164.304, Y  +696.571, Z    +0.000, E1   -14.525, E3 +376043.191}
SPL {X  -165.498, Y  +682.585, Z    +0.000, E1    -6.769, E3 +376042.866}
SPL {X  -165.650, Y  +674.975, Z    +0.000, E1    -1.888, E3 +376041.224}
SPL {X  -165.650, Y  +670.481, Z    +0.000, E1    +1.454, E3 +376040.665}
SPL {X  -165.650, Y  +665.304, Z    +0.000, E1    +6.303, E3 +376039.168}
SPL {X  -165.650, Y  +657.587, Z    +0.000, E1   +14.733, E3 +376037.942}
SPL {X  -165.650, Y  +646.511, Z    +0.000, E1   +26.434, E3 +376040.503}
SPL {X  -165.650, Y  +637.905, Z    +0.000, E1   +40.225, E3 +376028.628}
SPL {X  -165.650, Y  +611.479, Z    +0.000, E1   +52.226, E3 +376042.180}
SPL {X  -165.650, Y  +599.923, Z    +0.000, E1   +51.240, E3 +376059.269}
SPL {X  -165.650, Y  +553.219, Z    +0.000, E1   +52.865, E3 +376116.030}
ENDSPLINE

SPLINE
SPL {X  -165.650, Y  +569.883, Z    +0.000, E1   +45.183, E3 +376131.707}
ENDSPLINE

SPLINE
SPL {X  -165.650, Y  +561.960, Z    +0.000, E1   +45.285, E3 +376147.362}
SPL {X  -165.650, Y  +554.065, Z    +0.000, E1   +45.254, E3 +376163.424}
SPL {X  -165.650, Y  +548.074, Z    +0.000, E1   +45.245, E3 +376175.535}
SPL {X  -165.650, Y  +542.958, Z    +0.000, E1   +45.131, E3 +376186.665}
SPL {X  -165.650, Y  +535.288, Z    +0.000, E1   +45.332, E3 +376201.106}
SPL {X  -165.650, Y  +529.160, Z    +0.000, E1   +45.215, E3 +376214.087}
SPL {X  -165.650, Y  +522.672, Z    +0.000, E1   +45.331, E3 +376226.653}
SPL {X  -165.650, Y  +516.211, Z    +0.000, E1   +45.175, E3 +376240.613}
SPL {X  -165.650, Y  +509.762, Z    +0.000, E1   +45.191, E3 +376253.655}
SPL {X  -165.650, Y  +503.812, Z    +0.000, E1   +45.188, E3 +376265.694}
SPL {X  -165.650, Y  +499.646, Z    +0.000, E1   +44.886, E3 +376275.965}
ENDSPLINE

SPLINE
SPL {X  -165.650, Y  +514.834, Z    +0.000, E1   +36.829, E3 +376288.731}
ENDSPLINE

SPLINE
SPL {X  -165.650, Y  +506.421, Z    +0.000, E1   +37.886, E3 +376304.843}
SPL {X  -165.650, Y  +497.845, Z    +0.000, E1   +39.022, E3 +376320.006}
SPL {X  -165.650, Y  +488.971, Z    +0.000, E1   +40.149, E3 +376335.227}
SPL {X  -165.650, Y  +478.382, Z    +0.000, E1   +41.628, E3 +376351.424}
SPL {X  -165.650, Y  +468.596, Z    +0.000, E1   +42.673, E3 +376367.331}
SPL {X  -165.650, Y  +458.202, Z    +0.000, E1   +44.020, E3 +376381.872}
SPL {X  -165.650, Y  +452.111, Z    +0.000, E1   +44.272, E3 +376393.134}
ENDSPLINE

SPLINE
SPL {X  -165.650, Y  +459.414, Z    +0.000, E1   +39.996, E3 +376402.204}
ENDSPLINE

SPLINE
SPL {X  -165.650, Y  +455.681, Z    +0.000, E1   +39.641, E3 +376413.463}
SPL {X  -165.650, Y  +451.332, Z    +0.000, E1   +39.738, E3 +376423.596}
SPL {X  -165.650, Y  +448.050, Z    +0.000, E1   +39.392, E3 +376433.762}
SPL {X  -165.650, Y  +442.946, Z    +0.000, E1   +39.866, E3 +376443.536}
SPL {X  -165.650, Y  +439.091, Z    +0.000, E1   +39.674, E3 +376454.154}
SPL {X  -165.650, Y  +434.131, Z    +0.000, E1   +39.643, E3 +376466.667}
SPL {X  -165.650, Y  +428.810, Z    +0.000, E1   +39.691, E3 +376479.429}
SPL {X  -165.650, Y  +424.197, Z    +0.000, E1   +39.695, E3 +376490.788}
SPL {X  -165.650, Y  +420.220, Z    +0.000, E1   +39.526, E3 +376501.583}
SPL {X  -165.650, Y  +414.177, Z    +0.000, E1   +39.693, E3 +376515.710}
SPL {X  -165.650, Y  +407.394, Z    +0.000, E1   +39.797, E3 +376531.664}
SPL {X  -165.650, Y  +402.798, Z    +0.000, E1   +39.651, E3 +376543.786}
SPL {X  -165.650, Y  +398.253, Z    +0.000, E1   +39.688, E3 +376554.789}
SPL {X  -165.650, Y  +393.720, Z    +0.000, E1   +39.686, E3 +376565.964}
SPL {X  -165.650, Y  +389.210, Z    +0.000, E1   +39.696, E3 +376577.013}
SPL {X  -165.650, Y  +384.878, Z    +0.000, E1   +39.631, E3 +376588.090}
SPL {X  -165.650, Y  +378.931, Z    +0.000, E1   +39.598, E3 +376603.186}
SPL {X  -165.490, Y  +371.216, Z    +0.000, E1   +39.708, E3 +376621.558}
SPL {X  -165.055, Y  +364.469, Z    +0.000, E1   +39.623, E3 +376638.654}
SPL {X  -164.424, Y  +358.387, Z    +0.000, E1   +39.525, E3 +376654.177}
SPL {X  -163.775, Y  +353.645, Z    +0.000, E1   +39.313, E3 +376667.057}
SPL {X  -162.932, Y  +348.615, Z    +0.000, E1   +39.259, E3 +376679.821}
SPL {X  -161.858, Y  +343.258, Z    +0.000, E1   +39.040, E3 +376694.360}
SPL {X  -160.812, Y  +338.758, Z    +0.000, E1   +38.898, E3 +376706.085}
SPL {X  -159.926, Y  +335.332, Z    +0.000, E1   +38.809, E3 +376715.043}
SPL {X  -153.020, Y  +315.059, Z    +0.000, E1   +45.580, E3 +376721.774}
SPL {X  -148.632, Y  +305.368, Z    +0.000, E1   +40.700, E3 +376781.376}
SPL {X  -145.004, Y  +298.414, Z    +0.000, E1   +40.971, E3 +376806.111}
ENDSPLINE

SPLINE
SPL {X  -149.687, Y  +307.551, Z    +0.000, E1   +36.303, E3 +376841.543}
SPL {X  -158.807, Y  +331.381, Z    +0.000, E1   +26.928, E3 +376865.196}
SPL {X  -164.505, Y  +359.058, Z    +0.000, E1   +13.887, E3 +376853.958}
SPL {X  -165.494, Y  +371.321, Z    +0.000, E1    +7.176, E3 +376852.518}
SPL {X  -165.650, Y  +379.419, Z    +0.000, E1    +2.065, E3 +376850.200}
SPL {X  -165.650, Y  +383.176, Z    +0.000, E1    -0.610, E3 +376851.195}
SPL {X  -165.650, Y  +388.696, Z    +0.000, E1    -5.134, E3 +376849.471}
SPL {X  -165.650, Y  +394.663, Z    +0.000, E1   -10.843, E3 +376850.627}
SPL {X  -165.650, Y  +400.450, Z    +0.000, E1   -18.287, E3 +376841.926}
SPL {X  -165.650, Y  +409.248, Z    +0.000, E1   -26.478, E3 +376845.549}
SPL {X  -165.650, Y  +418.660, Z    +0.000, E1   -36.186, E3 +376843.025}
SPL {X  -165.650, Y  +444.260, Z    +0.000, E1   -47.328, E3 +376858.773}
SPL {X  -165.650, Y  +458.981, Z    +0.000, E1   -49.189, E3 +376874.317}
SPL {X  -165.650, Y  +493.049, Z    +0.000, E1   -51.657, E3 +376913.350}
ENDSPLINE

SPLINE
SPL {X  -165.650, Y  +468.984, Z    +0.000, E1   -41.461, E3 +376926.210}
SPL {X  -165.650, Y  +467.052, Z    +0.000, E1   -38.928, E3 +376936.825}
ENDSPLINE

SPLINE
SPL {X  -165.650, Y  +471.956, Z    +0.000, E1   -39.047, E3 +376948.476}
SPL {X  -165.650, Y  +476.270, Z    +0.000, E1   -39.142, E3 +376958.732}
SPL {X  -165.650, Y  +479.585, Z    +0.000, E1   -39.047, E3 +376967.643}
SPL {X  -165.650, Y  +484.115, Z    +0.000, E1   -39.050, E3 +376979.121}
SPL {X  -165.650, Y  +490.374, Z    +0.000, E1   -39.169, E3 +376994.241}
SPL {X  -165.650, Y  +496.519, Z    +0.000, E1   -39.062, E3 +377010.316}
SPL {X  -165.650, Y  +501.480, Z    +0.000, E1   -39.099, E3 +377022.473}
SPL {X  -165.650, Y  +505.989, Z    +0.000, E1   -39.067, E3 +377034.106}
SPL {X  -165.650, Y  +512.188, Z    +0.000, E1   -39.077, E3 +377049.749}
SPL {X  -165.650, Y  +518.439, Z    +0.000, E1   -39.071, E3 +377065.474}
SPL {X  -165.650, Y  +523.032, Z    +0.000, E1   -38.966, E3 +377077.609}
SPL {X  -165.650, Y  +527.474, Z    +0.000, E1   -39.169, E3 +377087.559}
SPL {X  -165.650, Y  +532.836, Z    +0.000, E1   -39.150, E3 +377101.342}
SPL {X  -165.650, Y  +539.651, Z    +0.000, E1   -39.087, E3 +377118.859}
SPL {X  -165.650, Y  +546.018, Z    +0.000, E1   -39.065, E3 +377134.984}
SPL {X  -165.650, Y  +551.666, Z    +0.000, E1   -39.102, E3 +377148.933}
SPL {X  -165.650, Y  +555.880, Z    +0.000, E1   -39.094, E3 +377159.505}
SPL {X  -165.650, Y  +559.255, Z    +0.000, E1   -39.167, E3 +377167.541}
SPL {X  -165.650, Y  +562.850, Z    +0.000, E1   -38.959, E3 +377177.938}
SPL {X  -165.650, Y  +568.257, Z    +0.000, E1   -39.077, E3 +377190.894}
SPL {X  -165.650, Y  +573.200, Z    +0.000, E1   -39.061, E3 +377203.428}
SPL {X  -165.650, Y  +578.240, Z    +0.000, E1   -39.117, E3 +377215.769}
SPL {X  -165.650, Y  +582.804, Z    +0.000, E1   -39.080, E3 +377227.476}
SPL {X  -165.650, Y  +587.640, Z    +0.000, E1   -39.069, E3 +377239.733}
SPL {X  -165.650, Y  +593.610, Z    +0.000, E1   -39.204, E3 +377254.007}
SPL {X  -165.650, Y  +599.021, Z    +0.000, E1   -38.950, E3 +377269.156}
SPL {X  -165.650, Y  +604.635, Z    +0.000, E1   -39.163, E3 +377281.933}
SPL {X  -165.650, Y  +608.365, Z    +0.000, E1   -39.063, E3 +377291.923}
SPL {X  -165.650, Y  +612.142, Z    +0.000, E1   -39.023, E3 +377301.653}
SPL {X  -165.650, Y  +616.635, Z    +0.000, E1   -39.260, E3 +377311.541}
SPL {X  -165.650, Y  +620.299, Z    +0.000, E1   -38.904, E3 +377322.927}
SPL {X  -165.650, Y  +625.662, Z    +0.000, E1   -39.189, E3 +377334.738}
SPL {X  -165.650, Y  +629.982, Z    +0.000, E1   -39.063, E3 +377346.340}
SPL {X  -165.650, Y  +635.019, Z    +0.000, E1   -39.106, E3 +377358.822}
SPL {X  -165.650, Y  +641.706, Z    +0.000, E1   -39.097, E3 +377375.889}
SPL {X  -165.650, Y  +648.294, Z    +0.000, E1   -39.142, E3 +377392.011}
SPL {X  -165.650, Y  +652.477, Z    +0.000, E1   -39.068, E3 +377402.913}
SPL {X  -165.650, Y  +656.920, Z    +0.000, E1   -39.120, E3 +377413.869}
SPL {X  -165.650, Y  +662.945, Z    +0.000, E1   -39.141, E3 +377428.974}
SPL {X  -165.650, Y  +668.296, Z    +0.000, E1   -39.077, E3 +377442.699}
SPL {X  -165.650, Y  +673.138, Z    +0.000, E1   -39.196, E3 +377454.155}
SPL {X  -165.640, Y  +677.281, Z    +0.000, E1   -38.803, E3 +377467.043}
SPL {X  -165.461, Y  +683.414, Z    +0.000, E1   -39.212, E3 +377480.027}
SPL {X  -165.139, Y  +688.497, Z    +0.000, E1   -39.013, E3 +377494.079}
SPL {X  -164.471, Y  +695.227, Z    +0.000, E1   -38.971, E3 +377511.374}
SPL {X  -163.525, Y  +701.945, Z    +0.000, E1   -38.769, E3 +377529.428}
SPL {X  -162.700, Y  +706.623, Z    +0.000, E1   -38.580, E3 +377542.103}
SPL {X  -161.983, Y  +710.160, Z    +0.000, E1   -38.439, E3 +377551.883}
SPL {X  -161.163, Y  +713.794, Z    +0.000, E1   -38.390, E3 +377561.252}
SPL {X  -160.158, Y  +717.801, Z    +0.000, E1   -38.225, E3 +377572.382}
SPL {X  -155.870, Y  +731.575, Z    +0.000, E1   -42.661, E3 +377579.845}
SPL {X  -137.799, Y  +767.431, Z    +0.000, E1   -46.550, E3 +377636.355}
ENDSPLINE

SPLINE
SPL {X  -141.948, Y  +760.885, Z    +0.000, E1   -42.258, E3 +377668.491}
SPL {X  -160.264, Y  +717.397, Z    +0.000, E1   -24.835, E3 +377709.676}
SPL {X  -164.762, Y  +692.628, Z    +0.000, E1   -12.660, E3 +377712.929}
SPL {X  -165.581, Y  +680.274, Z    +0.000, E1    -5.699, E3 +377708.413}
SPL {X  -165.650, Y  +672.825, Z    +0.000, E1    -0.909, E3 +377706.602}
SPL {X  -165.650, Y  +667.803, Z    +0.000, E1    +2.989, E3 +377706.062}
SPL {X  -165.650, Y  +662.773, Z    +0.000, E1    +7.549, E3 +377705.984}
SPL {X  -165.650, Y  +656.581, Z    +0.000, E1   +13.870, E3 +377704.033}
SPL {X  -165.650, Y  +648.120, Z    +0.000, E1   +22.794, E3 +377703.264}
SPL {X  -165.650, Y  +632.103, Z    +0.000, E1   +42.949, E3 +377690.222}
SPL {X  -165.650, Y  +608.448, Z    +0.000, E1   +47.265, E3 +377716.662}
SPL {X  -165.650, Y  +595.526, Z    +0.000, E1   +48.856, E3 +377730.520}
SPL {X  -165.650, Y  +568.828, Z    +0.000, E1   +48.639, E3 +377773.073}
ENDSPLINE

SPLINE
SPL {X  -165.650, Y  +586.972, Z    +0.000, E1   +40.422, E3 +377783.772}
ENDSPLINE

SPLINE
SPL {X  -165.650, Y  +585.370, Z    +0.000, E1   +38.910, E3 +377797.032}
SPL {X  -165.650, Y  +580.805, Z    +0.000, E1   +38.877, E3 +377808.654}
SPL {X  -165.650, Y  +575.679, Z    +0.000, E1   +38.947, E3 +377821.377}
SPL {X  -165.650, Y  +570.765, Z    +0.000, E1   +38.919, E3 +377833.818}
SPL {X  -165.650, Y  +566.463, Z    +0.000, E1   +38.933, E3 +377844.709}
SPL {X  -165.650, Y  +560.094, Z    +0.000, E1   +38.931, E3 +377861.030}
SPL {X  -165.650, Y  +554.358, Z    +0.000, E1   +38.887, E3 +377875.608}
SPL {X  -165.650, Y  +549.409, Z    +0.000, E1   +38.884, E3 +377888.289}
SPL {X  -165.650, Y  +544.480, Z    +0.000, E1   +38.998, E3 +377899.952}
SPL {X  -165.650, Y  +540.151, Z    +0.000, E1   +38.996, E3 +377910.998}
SPL {X  -165.650, Y  +534.008, Z    +0.000, E1   +38.962, E3 +377926.840}
SPL {X  -165.650, Y  +528.320, Z    +0.000, E1   +38.809, E3 +377942.076}
SPL {X  -165.650, Y  +522.377, Z    +0.000, E1   +38.974, E3 +377956.196}
ENDSPLINE

SPLINE
SPL {X  -165.650, Y  +539.854, Z    +0.000, E1   +28.090, E3 +377972.813}
ENDSPLINE

SPLINE
SPL {X  -165.650, Y  +534.443, Z    +0.000, E1   +28.969, E3 +377986.864}
SPL {X  -165.650, Y  +530.452, Z    +0.000, E1   +29.664, E3 +377996.597}
SPL {X  -165.650, Y  +523.712, Z    +0.000, E1   +30.911, E3 +378011.879}
SPL {X  -165.650, Y  +516.975, Z    +0.000, E1   +31.942, E3 +378027.473}
SPL {X  -165.650, Y  +512.706, Z    +0.000, E1   +32.573, E3 +378037.134}
SPL {X  -165.650, Y  +507.785, Z    +0.000, E1   +33.438, E3 +378047.072}
SPL {X  -165.650, Y  +501.257, Z    +0.000, E1   +34.478, E3 +378060.311}
SPL {X  -165.650, Y  +495.236, Z    +0.000, E1   +35.288, E3 +378072.817}
SPL {X  -165.650, Y  +488.684, Z    +0.000, E1   +36.217, E3 +378085.714}
SPL {X  -165.650, Y  +481.130, Z    +0.000, E1   +37.251, E3 +378100.023}
SPL {X  -165.650, Y  +475.455, Z    +0.000, E1   +37.964, E3 +378110.679}
SPL {X  -165.650, Y  +469.901, Z    +0.000, E1   +38.767, E3 +378120.173}
SPL {X  -165.650, Y  +465.276, Z    +0.000, E1   +39.067, E3 +378130.050}
SPL {X  -165.650, Y  +459.623, Z    +0.000, E1   +39.919, E3 +378138.986}
SPL {X  -165.650, Y  +455.681, Z    +0.000, E1   +39.641, E3 +378150.306}
SPL {X  -165.650, Y  +451.332, Z    +0.000, E1   +39.738, E3 +378160.438}
SPL {X  -165.650, Y  +448.050, Z    +0.000, E1   +39.392, E3 +378170.604}
SPL {X  -165.650, Y  +442.946, Z    +0.000, E1   +39.866, E3 +378180.378}
SPL {X  -165.650, Y  +439.091, Z    +0.000, E1   +39.674, E3 +378190.996}
SPL {X  -165.650, Y  +434.131, Z    +0.000, E1   +39.643, E3 +378203.509}
SPL {X  -165.650, Y  +428.810, Z    +0.000, E1   +39.691, E3 +378216.271}
SPL {X  -165.650, Y  +424.197, Z    +0.000, E1   +39.695, E3 +378227.630}
SPL {X  -165.650, Y  +420.220, Z    +0.000, E1   +39.526, E3 +378238.425}
SPL {X  -165.650, Y  +414.177, Z    +0.000, E1   +39.693, E3 +378252.552}
SPL {X  -165.650, Y  +407.394, Z    +0.000, E1   +39.797, E3 +378268.506}
SPL {X  -165.650, Y  +402.798, Z    +0.000, E1   +39.651, E3 +378280.628}
SPL {X  -165.650, Y  +398.253, Z    +0.000, E1   +39.688, E3 +378291.631}
SPL {X  -165.650, Y  +393.720, Z    +0.000, E1   +39.686, E3 +378302.806}
SPL {X  -165.650, Y  +389.210, Z    +0.000, E1   +39.696, E3 +378313.855}
SPL {X  -165.650, Y  +384.878, Z    +0.000, E1   +39.631, E3 +378324.932}
SPL {X  -165.650, Y  +378.931, Z    +0.000, E1   +39.598, E3 +378340.028}
SPL {X  -165.490, Y  +371.216, Z    +0.000, E1   +39.708, E3 +378358.400}
SPL {X  -165.216, Y  +366.519, Z    +0.000, E1   +39.498, E3 +378371.021}
SPL {X  -164.790, Y  +361.646, Z    +0.000, E1   +39.684, E3 +378382.015}
SPL {X  -164.317, Y  +357.530, Z    +0.000, E1   +39.402, E3 +378393.729}
SPL {X  -163.775, Y  +353.645, Z    +0.000, E1   +39.313, E3 +378403.899}
SPL {X  -162.932, Y  +348.615, Z    +0.000, E1   +39.259, E3 +378416.664}
SPL {X  -162.143, Y  +344.596, Z    +0.000, E1   +39.019, E3 +378427.880}
SPL {X  -161.093, Y  +339.912, Z    +0.000, E1   +38.966, E3 +378439.831}
SPL {X  -159.926, Y  +335.332, Z    +0.000, E1   +38.809, E3 +378451.885}
SPL {X  -153.020, Y  +315.059, Z    +0.000, E1   +45.580, E3 +378458.616}
SPL {X  -148.632, Y  +305.368, Z    +0.000, E1   +40.700, E3 +378518.218}
SPL {X  -145.004, Y  +298.414, Z    +0.000, E1   +40.971, E3 +378542.953}
ENDSPLINE

SPLINE
SPL {X  -149.687, Y  +307.551, Z    +0.000, E1   +36.303, E3 +378578.386}
SPL {X  -158.807, Y  +331.381, Z    +0.000, E1   +26.928, E3 +378602.038}
SPL {X  -164.505, Y  +359.058, Z    +0.000, E1   +13.887, E3 +378590.800}
SPL {X  -165.334, Y  +368.271, Z    +0.000, E1    +8.886, E3 +378588.638}
SPL {X  -165.596, Y  +374.277, Z    +0.000, E1    +5.306, E3 +378590.020}
SPL {X  -165.650, Y  +379.419, Z    +0.000, E1    +2.065, E3 +378587.042}
SPL {X  -165.650, Y  +383.176, Z    +0.000, E1    -0.610, E3 +378588.037}
SPL {X  -165.650, Y  +387.435, Z    +0.000, E1    -4.104, E3 +378586.397}
SPL {X  -165.650, Y  +393.422, Z    +0.000, E1    -9.605, E3 +378586.954}
SPL {X  -165.650, Y  +400.450, Z    +0.000, E1   -18.287, E3 +378578.769}
SPL {X  -165.650, Y  +409.248, Z    +0.000, E1   -26.478, E3 +378582.391}
SPL {X  -165.650, Y  +418.660, Z    +0.000, E1   -36.186, E3 +378579.868}
SPL {X  -165.650, Y  +444.260, Z    +0.000, E1   -47.328, E3 +378595.615}
SPL {X  -165.650, Y  +458.981, Z    +0.000, E1   -49.189, E3 +378611.159}
SPL {X  -165.650, Y  +493.049, Z    +0.000, E1   -51.657, E3 +378650.192}
ENDSPLINE

SPLINE
SPL {X  -165.650, Y  +468.984, Z    +0.000, E1   -41.461, E3 +378663.052}
SPL {X  -165.650, Y  +467.052, Z    +0.000, E1   -38.928, E3 +378673.667}
ENDSPLINE

SPLINE
SPL {X  -165.650, Y  +471.956, Z    +0.000, E1   -39.047, E3 +378685.318}
SPL {X  -165.650, Y  +476.270, Z    +0.000, E1   -39.142, E3 +378695.574}
SPL {X  -165.650, Y  +479.585, Z    +0.000, E1   -39.047, E3 +378704.486}
SPL {X  -165.650, Y  +484.115, Z    +0.000, E1   -39.050, E3 +378715.963}
SPL {X  -165.650, Y  +490.374, Z    +0.000, E1   -39.169, E3 +378731.083}
SPL {X  -165.650, Y  +495.141, Z    +0.000, E1   -39.109, E3 +378743.239}
SPL {X  -165.650, Y  +499.941, Z    +0.000, E1   -39.068, E3 +378755.768}
SPL {X  -165.650, Y  +505.989, Z    +0.000, E1   -39.067, E3 +378770.948}
SPL {X  -165.650, Y  +512.188, Z    +0.000, E1   -39.077, E3 +378786.591}
SPL {X  -165.650, Y  +516.634, Z    +0.000, E1   -39.035, E3 +378797.837}
SPL {X  -165.650, Y  +521.541, Z    +0.000, E1   -39.052, E3 +378810.383}
SPL {X  -165.650, Y  +527.474, Z    +0.000, E1   -39.169, E3 +378824.401}
SPL {X  -165.650, Y  +532.836, Z    +0.000, E1   -39.150, E3 +378838.184}
SPL {X  -165.650, Y  +537.667, Z    +0.000, E1   -38.986, E3 +378851.128}
SPL {X  -165.650, Y  +541.183, Z    +0.000, E1   -39.101, E3 +378859.316}
SPL {X  -165.650, Y  +546.018, Z    +0.000, E1   -39.065, E3 +378871.826}
SPL {X  -165.650, Y  +551.666, Z    +0.000, E1   -39.102, E3 +378885.775}
SPL {X  -165.650, Y  +557.612, Z    +0.000, E1   -39.166, E3 +378900.422}
SPL {X  -165.650, Y  +562.850, Z    +0.000, E1   -38.959, E3 +378914.780}
SPL {X  -165.650, Y  +568.257, Z    +0.000, E1   -39.077, E3 +378927.736}
SPL {X  -165.650, Y  +573.200, Z    +0.000, E1   -39.061, E3 +378940.270}
SPL {X  -165.650, Y  +578.240, Z    +0.000, E1   -39.117, E3 +378952.611}
SPL {X  -165.650, Y  +582.804, Z    +0.000, E1   -39.080, E3 +378964.319}
SPL {X  -165.650, Y  +587.640, Z    +0.000, E1   -39.069, E3 +378976.575}
SPL {X  -165.650, Y  +592.685, Z    +0.000, E1   -39.263, E3 +378988.040}
SPL {X  -165.650, Y  +596.539, Z    +0.000, E1   -39.049, E3 +378999.029}
SPL {X  -165.650, Y  +599.973, Z    +0.000, E1   -38.814, E3 +379009.082}
SPL {X  -165.650, Y  +604.635, Z    +0.000, E1   -39.163, E3 +379018.775}
SPL {X  -165.650, Y  +608.365, Z    +0.000, E1   -39.063, E3 +379028.765}
SPL {X  -165.650, Y  +613.618, Z    +0.000, E1   -39.137, E3 +379041.629}
SPL {X  -165.650, Y  +619.584, Z    +0.000, E1   -39.045, E3 +379057.266}
SPL {X  -165.650, Y  +625.662, Z    +0.000, E1   -39.189, E3 +379071.580}
SPL {X  -165.650, Y  +629.982, Z    +0.000, E1   -39.063, E3 +379083.182}
SPL {X  -165.650, Y  +635.019, Z    +0.000, E1   -39.106, E3 +379095.664}
SPL {X  -165.650, Y  +640.403, Z    +0.000, E1   -39.127, E3 +379109.059}
SPL {X  -165.650, Y  +643.707, Z    +0.000, E1   -38.911, E3 +379118.598}
SPL {X  -165.650, Y  +648.294, Z    +0.000, E1   -39.142, E3 +379128.853}
SPL {X  -165.650, Y  +652.477, Z    +0.000, E1   -39.068, E3 +379139.756}
SPL {X  -165.650, Y  +656.920, Z    +0.000, E1   -39.120, E3 +379150.711}
SPL {X  -165.650, Y  +662.945, Z    +0.000, E1   -39.141, E3 +379165.816}
SPL {X  -165.650, Y  +668.296, Z    +0.000, E1   -39.077, E3 +379179.541}
SPL {X  -165.650, Y  +673.138, Z    +0.000, E1   -39.196, E3 +379190.997}
SPL {X  -165.640, Y  +677.281, Z    +0.000, E1   -38.803, E3 +379203.885}
SPL {X  -165.461, Y  +683.414, Z    +0.000, E1   -39.212, E3 +379216.870}
SPL {X  -165.139, Y  +688.497, Z    +0.000, E1   -39.013, E3 +379230.921}
SPL {X  -164.471, Y  +695.227, Z    +0.000, E1   -38.971, E3 +379248.217}
SPL {X  -163.795, Y  +700.218, Z    +0.000, E1   -38.698, E3 +379262.163}
SPL {X  -162.937, Y  +705.358, Z    +0.000, E1   -38.703, E3 +379275.231}
SPL {X  -161.983, Y  +710.160, Z    +0.000, E1   -38.439, E3 +379288.725}
SPL {X  -160.874, Y  +714.989, Z    +0.000, E1   -38.205, E3 +379302.386}
SPL {X  -158.364, Y  +724.087, Z    +0.000, E1   -39.961, E3 +379314.592}
SPL {X  -138.706, Y  +766.057, Z    +0.000, E1   -46.957, E3 +379365.583}
ENDSPLINE

SPLINE
SPL {X  -141.948, Y  +760.885, Z    +0.000, E1   -42.258, E3 +379405.334}
SPL {X  -157.904, Y  +725.564, Z    +0.000, E1   -28.229, E3 +379448.585}
SPL {X  -161.595, Y  +711.926, Z    +0.000, E1   -22.341, E3 +379445.012}
SPL {X  -164.457, Y  +695.345, Z    +0.000, E1   -14.031, E3 +379453.460}
SPL {X  -165.312, Y  +686.072, Z    +0.000, E1    -9.096, E3 +379446.553}
SPL {X  -165.649, Y  +676.021, Z    +0.000, E1    -3.061, E3 +379443.982}
SPL {X  -165.650, Y  +671.288, Z    +0.000, E1    +0.282, E3 +379443.147}
SPL {X  -165.650, Y  +667.803, Z    +0.000, E1    +2.989, E3 +379442.904}
SPL {X  -165.650, Y  +662.773, Z    +0.000, E1    +7.549, E3 +379442.826}
SPL {X  -165.650, Y  +656.581, Z    +0.000, E1   +13.870, E3 +379440.875}
SPL {X  -165.650, Y  +648.120, Z    +0.000, E1   +22.794, E3 +379440.106}
SPL {X  -165.650, Y  +632.103, Z    +0.000, E1   +42.949, E3 +379427.064}
SPL {X  -165.650, Y  +608.448, Z    +0.000, E1   +47.265, E3 +379453.504}
SPL {X  -165.650, Y  +595.526, Z    +0.000, E1   +48.856, E3 +379467.362}
SPL {X  -165.650, Y  +568.828, Z    +0.000, E1   +48.639, E3 +379509.916}
ENDSPLINE

SPLINE
SPL {X  -165.650, Y  +586.972, Z    +0.000, E1   +40.422, E3 +379520.614}
ENDSPLINE

SPLINE
SPL {X  -165.650, Y  +585.370, Z    +0.000, E1   +38.910, E3 +379533.874}
SPL {X  -165.650, Y  +580.805, Z    +0.000, E1   +38.877, E3 +379545.496}
SPL {X  -165.650, Y  +575.679, Z    +0.000, E1   +38.947, E3 +379558.219}
SPL {X  -165.650, Y  +569.616, Z    +0.000, E1   +38.966, E3 +379573.377}
SPL {X  -165.650, Y  +564.364, Z    +0.000, E1   +38.909, E3 +379587.030}
SPL {X  -165.650, Y  +559.065, Z    +0.000, E1   +38.883, E3 +379600.608}
SPL {X  -165.650, Y  +554.358, Z    +0.000, E1   +38.887, E3 +379612.450}
SPL {X  -165.650, Y  +549.409, Z    +0.000, E1   +38.884, E3 +379625.131}
SPL {X  -165.650, Y  +542.772, Z    +0.000, E1   +39.054, E3 +379640.926}
SPL {X  -165.650, Y  +537.647, Z    +0.000, E1   +38.838, E3 +379655.089}
SPL {X  -165.650, Y  +532.636, Z    +0.000, E1   +39.009, E3 +379666.735}
SPL {X  -165.650, Y  +528.320, Z    +0.000, E1   +38.809, E3 +379678.918}
SPL {X  -165.650, Y  +522.377, Z    +0.000, E1   +38.974, E3 +379693.038}
ENDSPLINE

SPLINE
SPL {X  -165.650, Y  +539.854, Z    +0.000, E1   +28.090, E3 +379709.655}
ENDSPLINE

SPLINE
SPL {X  -165.650, Y  +534.443, Z    +0.000, E1   +28.969, E3 +379723.706}
SPL {X  -165.650, Y  +530.452, Z    +0.000, E1   +29.664, E3 +379733.440}
SPL {X  -165.650, Y  +525.298, Z    +0.000, E1   +30.602, E3 +379745.250}
SPL {X  -165.650, Y  +518.290, Z    +0.000, E1   +31.783, E3 +379761.142}
SPL {X  -165.650, Y  +512.706, Z    +0.000, E1   +32.573, E3 +379773.977}
SPL {X  -165.650, Y  +507.785, Z    +0.000, E1   +33.438, E3 +379783.914}
SPL {X  -165.650, Y  +502.877, Z    +0.000, E1   +34.230, E3 +379793.802}
SPL {X  -165.650, Y  +496.704, Z    +0.000, E1   +35.113, E3 +379806.595}
SPL {X  -165.650, Y  +488.684, Z    +0.000, E1   +36.217, E3 +379822.556}
SPL {X  -165.650, Y  +481.130, Z    +0.000, E1   +37.251, E3 +379836.865}
SPL {X  -165.650, Y  +475.455, Z    +0.000, E1   +37.964, E3 +379847.521}
SPL {X  -165.650, Y  +469.901, Z    +0.000, E1   +38.767, E3 +379857.015}
SPL {X  -165.650, Y  +461.805, Z    +0.000, E1   +39.619, E3 +379872.358}
SPL {X  -165.650, Y  +455.681, Z    +0.000, E1   +39.641, E3 +379887.148}
SPL {X  -165.650, Y  +451.332, Z    +0.000, E1   +39.738, E3 +379897.280}
SPL {X  -165.650, Y  +448.050, Z    +0.000, E1   +39.392, E3 +379907.446}
SPL {X  -165.650, Y  +442.946, Z    +0.000, E1   +39.866, E3 +379917.220}
SPL {X  -165.650, Y  +439.091, Z    +0.000, E1   +39.674, E3 +379927.838}
SPL {X  -165.650, Y  +435.404, Z    +0.000, E1   +39.549, E3 +379937.675}
SPL {X  -165.650, Y  +429.757, Z    +0.000, E1   +39.737, E3 +379950.624}
SPL {X  -165.650, Y  +424.197, Z    +0.000, E1   +39.695, E3 +379964.472}
SPL {X  -165.650, Y  +420.220, Z    +0.000, E1   +39.526, E3 +379975.267}
SPL {X  -165.650, Y  +415.675, Z    +0.000, E1   +39.706, E3 +379985.428}
SPL {X  -165.650, Y  +410.648, Z    +0.000, E1   +39.653, E3 +379998.229}
SPL {X  -165.650, Y  +403.851, Z    +0.000, E1   +39.774, E3 +380014.315}
SPL {X  -165.650, Y  +398.253, Z    +0.000, E1   +39.688, E3 +380028.474}
SPL {X  -165.650, Y  +393.720, Z    +0.000, E1   +39.686, E3 +380039.648}
SPL {X  -165.650, Y  +389.210, Z    +0.000, E1   +39.696, E3 +380050.697}
SPL {X  -165.650, Y  +384.878, Z    +0.000, E1   +39.631, E3 +380061.774}
SPL {X  -165.650, Y  +378.931, Z    +0.000, E1   +39.598, E3 +380076.870}
SPL {X  -165.490, Y  +371.216, Z    +0.000, E1   +39.708, E3 +380095.242}
SPL {X  -165.216, Y  +366.519, Z    +0.000, E1   +39.498, E3 +380107.863}
SPL {X  -164.790, Y  +361.646, Z    +0.000, E1   +39.684, E3 +380118.857}
SPL {X  -164.317, Y  +357.530, Z    +0.000, E1   +39.402, E3 +380130.571}
SPL {X  -163.775, Y  +353.645, Z    +0.000, E1   +39.313, E3 +380140.741}
SPL {X  -162.932, Y  +348.615, Z    +0.000, E1   +39.259, E3 +380153.506}
SPL {X  -162.143, Y  +344.596, Z    +0.000, E1   +39.019, E3 +380164.722}
SPL {X  -161.093, Y  +339.912, Z    +0.000, E1   +38.966, E3 +380176.673}
SPL {X  -159.926, Y  +335.332, Z    +0.000, E1   +38.809, E3 +380188.727}
SPL {X  -153.020, Y  +315.059, Z    +0.000, E1   +45.580, E3 +380195.458}
SPL {X  -148.632, Y  +305.368, Z    +0.000, E1   +40.700, E3 +380255.060}
SPL {X  -145.004, Y  +298.414, Z    +0.000, E1   +40.971, E3 +380279.795}
ENDSPLINE

SPLINE
SPL {X  -149.687, Y  +307.551, Z    +0.000, E1   +36.303, E3 +380315.228}
SPL {X  -158.807, Y  +331.381, Z    +0.000, E1   +26.928, E3 +380338.880}
SPL {X  -164.505, Y  +359.058, Z    +0.000, E1   +13.887, E3 +380327.642}
SPL {X  -165.494, Y  +371.321, Z    +0.000, E1    +7.176, E3 +380326.202}
SPL {X  -165.650, Y  +379.419, Z    +0.000, E1    +2.065, E3 +380323.884}
SPL {X  -165.650, Y  +383.176, Z    +0.000, E1    -0.610, E3 +380324.879}
SPL {X  -165.650, Y  +387.435, Z    +0.000, E1    -4.104, E3 +380323.239}
SPL {X  -165.650, Y  +393.422, Z    +0.000, E1    -9.605, E3 +380323.796}
SPL {X  -165.650, Y  +400.450, Z    +0.000, E1   -18.287, E3 +380315.611}
SPL {X  -165.650, Y  +409.248, Z    +0.000, E1   -26.478, E3 +380319.234}
SPL {X  -165.650, Y  +418.660, Z    +0.000, E1   -36.186, E3 +380316.710}
SPL {X  -165.650, Y  +444.260, Z    +0.000, E1   -47.328, E3 +380332.457}
SPL {X  -165.650, Y  +458.981, Z    +0.000, E1   -49.189, E3 +380348.001}
SPL {X  -165.650, Y  +493.049, Z    +0.000, E1   -51.657, E3 +380387.034}
ENDSPLINE

SPLINE
SPL {X  -165.650, Y  +468.984, Z    +0.000, E1   -41.461, E3 +380399.894}
SPL {X  -165.650, Y  +467.052, Z    +0.000, E1   -38.928, E3 +380410.509}
ENDSPLINE

SPLINE
SPL {X  -165.650, Y  +471.956, Z    +0.000, E1   -39.047, E3 +380422.160}
SPL {X  -165.650, Y  +476.270, Z    +0.000, E1   -39.142, E3 +380432.416}
SPL {X  -165.650, Y  +480.876, Z    +0.000, E1   -39.050, E3 +380444.698}
SPL {X  -165.650, Y  +487.054, Z    +0.000, E1   -39.118, E3 +380459.837}
SPL {X  -165.650, Y  +491.785, Z    +0.000, E1   -39.157, E3 +380471.386}
SPL {X  -165.650, Y  +496.519, Z    +0.000, E1   -39.062, E3 +380484.001}
SPL {X  -165.650, Y  +502.351, Z    +0.000, E1   -39.056, E3 +380498.723}
SPL {X  -165.650, Y  +508.180, Z    +0.000, E1   -39.157, E3 +380512.789}
SPL {X  -165.650, Y  +514.341, Z    +0.000, E1   -39.047, E3 +380529.041}
SPL {X  -165.650, Y  +521.541, Z    +0.000, E1   -39.052, E3 +380547.225}
SPL {X  -165.650, Y  +528.401, Z    +0.000, E1   -39.135, E3 +380563.894}
SPL {X  -165.650, Y  +533.857, Z    +0.000, E1   -39.163, E3 +380577.399}
SPL {X  -165.650, Y  +539.651, Z    +0.000, E1   -39.087, E3 +380592.543}
SPL {X  -165.650, Y  +546.018, Z    +0.000, E1   -39.065, E3 +380608.668}
SPL {X  -165.650, Y  +551.666, Z    +0.000, E1   -39.102, E3 +380622.618}
SPL {X  -165.650, Y  +557.612, Z    +0.000, E1   -39.166, E3 +380637.264}
SPL {X  -165.650, Y  +562.850, Z    +0.000, E1   -38.959, E3 +380651.623}
SPL {X  -165.650, Y  +568.257, Z    +0.000, E1   -39.077, E3 +380664.578}
SPL {X  -165.650, Y  +573.200, Z    +0.000, E1   -39.061, E3 +380677.113}
SPL {X  -165.650, Y  +578.240, Z    +0.000, E1   -39.117, E3 +380689.453}
SPL {X  -165.650, Y  +582.804, Z    +0.000, E1   -39.080, E3 +380701.161}
SPL {X  -165.650, Y  +587.640, Z    +0.000, E1   -39.069, E3 +380713.417}
SPL {X  -165.650, Y  +592.685, Z    +0.000, E1   -39.263, E3 +380724.882}
SPL {X  -165.650, Y  +596.539, Z    +0.000, E1   -39.049, E3 +380735.871}
SPL {X  -165.650, Y  +599.973, Z    +0.000, E1   -38.814, E3 +380745.924}
SPL {X  -165.650, Y  +604.635, Z    +0.000, E1   -39.163, E3 +380755.617}
SPL {X  -165.650, Y  +608.365, Z    +0.000, E1   -39.063, E3 +380765.608}
SPL {X  -165.650, Y  +613.618, Z    +0.000, E1   -39.137, E3 +380778.472}
SPL {X  -165.650, Y  +619.584, Z    +0.000, E1   -39.045, E3 +380794.109}
SPL {X  -165.650, Y  +625.662, Z    +0.000, E1   -39.189, E3 +380808.422}
SPL {X  -165.650, Y  +629.982, Z    +0.000, E1   -39.063, E3 +380820.024}
SPL {X  -165.650, Y  +634.317, Z    +0.000, E1   -39.239, E3 +380829.814}
SPL {X  -165.650, Y  +639.215, Z    +0.000, E1   -39.074, E3 +380843.339}
SPL {X  -165.650, Y  +645.443, Z    +0.000, E1   -39.032, E3 +380859.207}
SPL {X  -165.650, Y  +651.452, Z    +0.000, E1   -39.128, E3 +380873.776}
SPL {X  -165.650, Y  +656.920, Z    +0.000, E1   -39.120, E3 +380887.553}
SPL {X  -165.650, Y  +661.125, Z    +0.000, E1   -39.092, E3 +380898.202}
SPL {X  -165.650, Y  +664.437, Z    +0.000, E1   -39.114, E3 +380906.410}
SPL {X  -165.650, Y  +668.296, Z    +0.000, E1   -39.077, E3 +380916.383}
SPL {X  -165.650, Y  +673.138, Z    +0.000, E1   -39.196, E3 +380927.839}
SPL {X  -165.640, Y  +677.281, Z    +0.000, E1   -38.803, E3 +380940.727}
SPL {X  -165.461, Y  +683.414, Z    +0.000, E1   -39.212, E3 +380953.712}
SPL {X  -165.139, Y  +688.497, Z    +0.000, E1   -39.013, E3 +380967.763}
SPL {X  -164.582, Y  +694.282, Z    +0.000, E1   -38.975, E3 +380982.511}
SPL {X  -163.926, Y  +699.336, Z    +0.000, E1   -38.767, E3 +380996.489}
SPL {X  -163.214, Y  +703.806, Z    +0.000, E1   -38.755, E3 +381007.675}
SPL {X  -162.700, Y  +706.623, Z    +0.000, E1   -38.580, E3 +381015.787}
SPL {X  -161.983, Y  +710.160, Z    +0.000, E1   -38.439, E3 +381025.567}
SPL {X  -161.163, Y  +713.794, Z    +0.000, E1   -38.390, E3 +381034.936}
SPL {X  -160.158, Y  +717.801, Z    +0.000, E1   -38.225, E3 +381046.066}
SPL {X  -155.870, Y  +731.575, Z    +0.000, E1   -42.661, E3 +381053.529}
SPL {X  -137.799, Y  +767.431, Z    +0.000, E1   -46.550, E3 +381110.039}
ENDSPLINE

SPLINE
SPL {X  -141.948, Y  +760.885, Z    +0.000, E1   -42.258, E3 +381142.176}
SPL {X  -160.264, Y  +717.397, Z    +0.000, E1   -24.835, E3 +381183.360}
SPL {X  -164.762, Y  +692.628, Z    +0.000, E1   -12.660, E3 +381186.613}
SPL {X  -165.581, Y  +680.274, Z    +0.000, E1    -5.699, E3 +381182.097}
SPL {X  -165.650, Y  +672.825, Z    +0.000, E1    -0.909, E3 +381180.286}
SPL {X  -165.650, Y  +667.803, Z    +0.000, E1    +2.989, E3 +381179.746}
SPL {X  -165.650, Y  +662.773, Z    +0.000, E1    +7.549, E3 +381179.668}
SPL {X  -165.650, Y  +656.581, Z    +0.000, E1   +13.870, E3 +381177.718}
SPL {X  -165.650, Y  +648.120, Z    +0.000, E1   +22.794, E3 +381176.949}
SPL {X  -165.650, Y  +632.103, Z    +0.000, E1   +42.949, E3 +381163.906}
SPL {X  -165.650, Y  +608.448, Z    +0.000, E1   +47.265, E3 +381190.346}
SPL {X  -165.650, Y  +595.526, Z    +0.000, E1   +48.856, E3 +381204.204}
SPL {X  -165.650, Y  +568.828, Z    +0.000, E1   +48.639, E3 +381246.758}
ENDSPLINE

SPLINE
SPL {X  -165.650, Y  +586.972, Z    +0.000, E1   +40.422, E3 +381257.456}
ENDSPLINE

SPLINE
SPL {X  -165.650, Y  +585.370, Z    +0.000, E1   +38.910, E3 +381270.716}
SPL {X  -165.650, Y  +580.805, Z    +0.000, E1   +38.877, E3 +381282.338}
SPL {X  -165.650, Y  +576.923, Z    +0.000, E1   +38.908, E3 +381292.016}
SPL {X  -165.650, Y  +571.957, Z    +0.000, E1   +38.951, E3 +381304.421}
SPL {X  -165.650, Y  +566.463, Z    +0.000, E1   +38.933, E3 +381318.393}
SPL {X  -165.650, Y  +561.565, Z    +0.000, E1   +38.903, E3 +381330.966}
SPL {X  -165.650, Y  +557.881, Z    +0.000, E1   +38.850, E3 +381340.541}
SPL {X  -165.650, Y  +552.770, Z    +0.000, E1   +38.963, E3 +381353.011}
SPL {X  -165.650, Y  +546.277, Z    +0.000, E1   +38.910, E3 +381369.753}
SPL {X  -165.650, Y  +540.151, Z    +0.000, E1   +38.996, E3 +381384.682}
SPL {X  -165.650, Y  +534.008, Z    +0.000, E1   +38.962, E3 +381400.524}
SPL {X  -165.650, Y  +528.320, Z    +0.000, E1   +38.809, E3 +381415.760}
SPL {X  -165.650, Y  +522.377, Z    +0.000, E1   +38.974, E3 +381429.880}
ENDSPLINE

SPLINE
SPL {X  -165.650, Y  +541.168, Z    +0.000, E1   +27.957, E3 +381442.220}
ENDSPLINE

SPLINE
SPL {X  -165.650, Y  +536.052, Z    +0.000, E1   +28.653, E3 +381456.855}
SPL {X  -165.650, Y  +530.452, Z    +0.000, E1   +29.664, E3 +381470.282}
SPL {X  -165.650, Y  +525.298, Z    +0.000, E1   +30.602, E3 +381482.092}
SPL {X  -165.650, Y  +518.290, Z    +0.000, E1   +31.783, E3 +381497.984}
SPL {X  -165.650, Y  +512.706, Z    +0.000, E1   +32.573, E3 +381510.819}
SPL {X  -165.650, Y  +507.785, Z    +0.000, E1   +33.438, E3 +381520.756}
SPL {X  -165.650, Y  +502.877, Z    +0.000, E1   +34.230, E3 +381530.644}
SPL {X  -165.650, Y  +499.289, Z    +0.000, E1   +34.735, E3 +381538.112}
SPL {X  -165.650, Y  +493.800, Z    +0.000, E1   +35.486, E3 +381549.483}
SPL {X  -165.650, Y  +485.583, Z    +0.000, E1   +36.670, E3 +381565.207}
SPL {X  -165.650, Y  +477.375, Z    +0.000, E1   +37.747, E3 +381580.726}
SPL {X  -165.650, Y  +469.901, Z    +0.000, E1   +38.767, E3 +381593.857}
SPL {X  -165.650, Y  +461.805, Z    +0.000, E1   +39.619, E3 +381609.201}
SPL {X  -165.650, Y  +455.681, Z    +0.000, E1   +39.641, E3 +381623.990}
SPL {X  -165.650, Y  +451.332, Z    +0.000, E1   +39.738, E3 +381634.122}
SPL {X  -165.650, Y  +448.050, Z    +0.000, E1   +39.392, E3 +381644.288}
SPL {X  -165.650, Y  +442.946, Z    +0.000, E1   +39.866, E3 +381654.062}
SPL {X  -165.650, Y  +439.091, Z    +0.000, E1   +39.674, E3 +381664.680}
SPL {X  -165.650, Y  +434.131, Z    +0.000, E1   +39.643, E3 +381677.193}
SPL {X  -165.650, Y  +428.810, Z    +0.000, E1   +39.691, E3 +381689.955}
SPL {X  -165.650, Y  +424.197, Z    +0.000, E1   +39.695, E3 +381701.314}
SPL {X  -165.650, Y  +420.220, Z    +0.000, E1   +39.526, E3 +381712.109}
SPL {X  -165.650, Y  +415.675, Z    +0.000, E1   +39.706, E3 +381722.271}
SPL {X  -165.650, Y  +410.648, Z    +0.000, E1   +39.653, E3 +381735.071}
SPL {X  -165.650, Y  +403.851, Z    +0.000, E1   +39.774, E3 +381751.157}
SPL {X  -165.650, Y  +398.253, Z    +0.000, E1   +39.688, E3 +381765.316}
SPL {X  -165.650, Y  +393.720, Z    +0.000, E1   +39.686, E3 +381776.490}
SPL {X  -165.650, Y  +389.210, Z    +0.000, E1   +39.696, E3 +381787.539}
SPL {X  -165.650, Y  +384.878, Z    +0.000, E1   +39.631, E3 +381798.616}
SPL {X  -165.650, Y  +380.529, Z    +0.000, E1   +39.528, E3 +381810.002}
SPL {X  -165.618, Y  +375.240, Z    +0.000, E1   +39.617, E3 +381822.597}
SPL {X  -165.428, Y  +369.922, Z    +0.000, E1   +39.705, E3 +381835.138}
SPL {X  -165.216, Y  +366.519, Z    +0.000, E1   +39.498, E3 +381844.705}
SPL {X  -164.790, Y  +361.646, Z    +0.000, E1   +39.684, E3 +381855.699}
SPL {X  -164.317, Y  +357.530, Z    +0.000, E1   +39.402, E3 +381867.413}
SPL {X  -163.775, Y  +353.645, Z    +0.000, E1   +39.313, E3 +381877.584}
SPL {X  -163.109, Y  +349.595, Z    +0.000, E1   +39.290, E3 +381887.645}
SPL {X  -162.309, Y  +345.398, Z    +0.000, E1   +39.085, E3 +381899.309}
SPL {X  -161.467, Y  +341.510, Z    +0.000, E1   +38.980, E3 +381909.354}
SPL {X  -160.812, Y  +338.758, Z    +0.000, E1   +38.898, E3 +381916.611}
SPL {X  -159.926, Y  +335.332, Z    +0.000, E1   +38.809, E3 +381925.569}
SPL {X  -153.020, Y  +315.059, Z    +0.000, E1   +45.580, E3 +381932.300}
SPL {X  -148.632, Y  +305.368, Z    +0.000, E1   +40.700, E3 +381991.902}
SPL {X  -145.004, Y  +298.414, Z    +0.000, E1   +40.971, E3 +382016.637}
ENDSPLINE

SPLINE
SPL {X  -149.687, Y  +307.551, Z    +0.000, E1   +36.303, E3 +382052.070}
SPL {X  -158.807, Y  +331.381, Z    +0.000, E1   +26.928, E3 +382075.722}
SPL {X  -164.505, Y  +359.058, Z    +0.000, E1   +13.887, E3 +382064.484}
SPL {X  -165.494, Y  +371.321, Z    +0.000, E1    +7.176, E3 +382063.044}
SPL {X  -165.650, Y  +379.419, Z    +0.000, E1    +2.065, E3 +382060.726}
SPL {X  -165.650, Y  +383.176, Z    +0.000, E1    -0.610, E3 +382061.721}
SPL {X  -165.650, Y  +387.435, Z    +0.000, E1    -4.104, E3 +382060.081}
SPL {X  -165.650, Y  +393.422, Z    +0.000, E1    -9.605, E3 +382060.638}
SPL {X  -165.650, Y  +400.450, Z    +0.000, E1   -18.287, E3 +382052.453}
SPL {X  -165.650, Y  +409.248, Z    +0.000, E1   -26.478, E3 +382056.076}
SPL {X  -165.650, Y  +418.660, Z    +0.000, E1   -36.186, E3 +382053.552}
SPL {X  -165.650, Y  +444.260, Z    +0.000, E1   -47.328, E3 +382069.299}
SPL {X  -165.650, Y  +458.981, Z    +0.000, E1   -49.189, E3 +382084.843}
SPL {X  -165.650, Y  +493.049, Z    +0.000, E1   -51.657, E3 +382123.876}
ENDSPLINE

SPLINE
SPL {X  -165.650, Y  +468.984, Z    +0.000, E1   -41.461, E3 +382136.736}
SPL {X  -165.650, Y  +467.052, Z    +0.000, E1   -38.928, E3 +382147.351}
ENDSPLINE

SPLINE
SPL {X  -165.650, Y  +471.956, Z    +0.000, E1   -39.047, E3 +382159.002}
SPL {X  -165.650, Y  +476.270, Z    +0.000, E1   -39.142, E3 +382169.258}
SPL {X  -165.650, Y  +479.585, Z    +0.000, E1   -39.047, E3 +382178.170}
SPL {X  -165.650, Y  +484.115, Z    +0.000, E1   -39.050, E3 +382189.648}
SPL {X  -165.650, Y  +490.374, Z    +0.000, E1   -39.169, E3 +382204.767}
SPL {X  -165.650, Y  +496.519, Z    +0.000, E1   -39.062, E3 +382220.843}
SPL {X  -165.650, Y  +502.351, Z    +0.000, E1   -39.056, E3 +382235.565}
SPL {X  -165.650, Y  +508.180, Z    +0.000, E1   -39.157, E3 +382249.631}
SPL {X  -165.650, Y  +513.074, Z    +0.000, E1   -38.997, E3 +382262.849}
SPL {X  -165.650, Y  +518.439, Z    +0.000, E1   -39.071, E3 +382276.000}
SPL {X  -165.650, Y  +523.032, Z    +0.000, E1   -38.966, E3 +382288.136}
SPL {X  -165.650, Y  +528.401, Z    +0.000, E1   -39.135, E3 +382300.736}
SPL {X  -165.650, Y  +533.857, Z    +0.000, E1   -39.163, E3 +382314.241}
SPL {X  -165.650, Y  +539.651, Z    +0.000, E1   -39.087, E3 +382329.385}
SPL {X  -165.650, Y  +544.603, Z    +0.000, E1   -39.103, E3 +382341.561}
SPL {X  -165.650, Y  +547.280, Z    +0.000, E1   -38.965, E3 +382349.141}
SPL {X  -165.650, Y  +551.666, Z    +0.000, E1   -39.102, E3 +382359.460}
SPL {X  -165.650, Y  +555.880, Z    +0.000, E1   -39.094, E3 +382370.031}
SPL {X  -165.650, Y  +559.255, Z    +0.000, E1   -39.167, E3 +382378.067}
SPL {X  -165.650, Y  +562.850, Z    +0.000, E1   -38.959, E3 +382388.465}
SPL {X  -165.650, Y  +568.257, Z    +0.000, E1   -39.077, E3 +382401.420}
SPL {X  -165.650, Y  +573.200, Z    +0.000, E1   -39.061, E3 +382413.955}
SPL {X  -165.650, Y  +578.240, Z    +0.000, E1   -39.117, E3 +382426.296}
SPL {X  -165.650, Y  +582.804, Z    +0.000, E1   -39.080, E3 +382438.003}
SPL {X  -165.650, Y  +587.640, Z    +0.000, E1   -39.069, E3 +382450.259}
SPL {X  -165.650, Y  +593.610, Z    +0.000, E1   -39.204, E3 +382464.533}
SPL {X  -165.650, Y  +599.021, Z    +0.000, E1   -38.950, E3 +382479.683}
SPL {X  -165.650, Y  +604.635, Z    +0.000, E1   -39.163, E3 +382492.459}
SPL {X  -165.650, Y  +608.365, Z    +0.000, E1   -39.063, E3 +382502.450}
SPL {X  -165.650, Y  +612.142, Z    +0.000, E1   -39.023, E3 +382512.180}
SPL {X  -165.650, Y  +616.635, Z    +0.000, E1   -39.260, E3 +382522.067}
SPL {X  -165.650, Y  +620.299, Z    +0.000, E1   -38.904, E3 +382533.453}
SPL {X  -165.650, Y  +625.662, Z    +0.000, E1   -39.189, E3 +382545.264}
SPL {X  -165.650, Y  +629.982, Z    +0.000, E1   -39.063, E3 +382556.866}
SPL {X  -165.650, Y  +634.317, Z    +0.000, E1   -39.239, E3 +382566.656}
SPL {X  -165.650, Y  +639.215, Z    +0.000, E1   -39.074, E3 +382580.182}
SPL {X  -165.650, Y  +643.707, Z    +0.000, E1   -38.911, E3 +382592.282}
SPL {X  -165.650, Y  +648.294, Z    +0.000, E1   -39.142, E3 +382602.537}
SPL {X  -165.650, Y  +652.477, Z    +0.000, E1   -39.068, E3 +382613.440}
SPL {X  -165.650, Y  +656.920, Z    +0.000, E1   -39.120, E3 +382624.395}
SPL {X  -165.650, Y  +662.945, Z    +0.000, E1   -39.141, E3 +382639.500}
SPL {X  -165.650, Y  +668.296, Z    +0.000, E1   -39.077, E3 +382653.225}
SPL {X  -165.650, Y  +674.193, Z    +0.000, E1   -39.034, E3 +382668.567}
SPL {X  -165.521, Y  +682.029, Z    +0.000, E1   -39.160, E3 +382687.535}
SPL {X  -165.241, Y  +687.126, Z    +0.000, E1   -39.221, E3 +382699.696}
SPL {X  -164.948, Y  +690.736, Z    +0.000, E1   -38.951, E3 +382710.549}
SPL {X  -164.363, Y  +696.109, Z    +0.000, E1   -38.853, E3 +382724.639}
SPL {X  -163.795, Y  +700.218, Z    +0.000, E1   -38.698, E3 +382735.847}
SPL {X  -162.937, Y  +705.358, Z    +0.000, E1   -38.703, E3 +382748.915}
SPL {X  -161.983, Y  +710.160, Z    +0.000, E1   -38.439, E3 +382762.409}
SPL {X  -161.163, Y  +713.794, Z    +0.000, E1   -38.390, E3 +382771.779}
SPL {X  -160.616, Y  +716.027, Z    +0.000, E1   -37.944, E3 +382779.981}
SPL {X  -158.364, Y  +724.087, Z    +0.000, E1   -39.961, E3 +382788.276}
SPL {X  -138.706, Y  +766.057, Z    +0.000, E1   -46.957, E3 +382839.268}
ENDSPLINE

SPLINE
SPL {X  -141.948, Y  +760.885, Z    +0.000, E1   -42.258, E3 +382879.018}
SPL {X  -152.484, Y  +740.219, Z    +0.000, E1   -33.928, E3 +382916.171}
SPL {X  -161.203, Y  +713.624, Z    +0.000, E1   -23.097, E3 +382920.587}
SPL {X  -164.762, Y  +692.628, Z    +0.000, E1   -12.660, E3 +382923.455}
SPL {X  -165.581, Y  +680.274, Z    +0.000, E1    -5.699, E3 +382918.940}
SPL {X  -165.650, Y  +674.578, Z    +0.000, E1    -2.045, E3 +382917.467}
SPL {X  -165.650, Y  +670.589, Z    +0.000, E1    +0.778, E3 +382916.904}
SPL {X  -165.650, Y  +666.842, Z    +0.000, E1    +3.871, E3 +382916.365}
SPL {X  -165.650, Y  +661.513, Z    +0.000, E1    +8.695, E3 +382916.273}
SPL {X  -165.650, Y  +654.973, Z    +0.000, E1   +15.752, E3 +382913.679}
SPL {X  -165.650, Y  +648.120, Z    +0.000, E1   +22.794, E3 +382913.791}
SPL {X  -165.650, Y  +632.103, Z    +0.000, E1   +42.949, E3 +382900.749}
SPL {X  -165.650, Y  +609.948, Z    +0.000, E1   +49.636, E3 +382918.175}
SPL {X  -165.650, Y  +601.895, Z    +0.000, E1   +47.595, E3 +382935.845}
SPL {X  -165.650, Y  +568.828, Z    +0.000, E1   +48.639, E3 +382983.600}
ENDSPLINE

SPLINE
SPL {X  -165.650, Y  +586.972, Z    +0.000, E1   +40.422, E3 +382994.299}
ENDSPLINE

SPLINE
SPL {X  -165.650, Y  +585.370, Z    +0.000, E1   +38.910, E3 +383007.559}
SPL {X  -165.650, Y  +580.805, Z    +0.000, E1   +38.877, E3 +383019.181}
SPL {X  -165.650, Y  +576.923, Z    +0.000, E1   +38.908, E3 +383028.858}
SPL {X  -165.650, Y  +571.957, Z    +0.000, E1   +38.951, E3 +383041.263}
SPL {X  -165.650, Y  +566.463, Z    +0.000, E1   +38.933, E3 +383055.235}
SPL {X  -165.650, Y  +561.565, Z    +0.000, E1   +38.903, E3 +383067.808}
SPL {X  -165.650, Y  +557.881, Z    +0.000, E1   +38.850, E3 +383077.383}
SPL {X  -165.650, Y  +552.770, Z    +0.000, E1   +38.963, E3 +383089.853}
SPL {X  -165.650, Y  +546.277, Z    +0.000, E1   +38.910, E3 +383106.595}
SPL {X  -165.650, Y  +540.151, Z    +0.000, E1   +38.996, E3 +383121.524}
SPL {X  -165.650, Y  +534.008, Z    +0.000, E1   +38.962, E3 +383137.366}
SPL {X  -165.650, Y  +528.320, Z    +0.000, E1   +38.809, E3 +383152.603}
SPL {X  -165.650, Y  +522.377, Z    +0.000, E1   +38.974, E3 +383166.722}
ENDSPLINE

SPLINE
SPL {X  -165.650, Y  +541.168, Z    +0.000, E1   +27.957, E3 +383179.062}
ENDSPLINE

SPLINE
SPL {X  -165.650, Y  +536.052, Z    +0.000, E1   +28.653, E3 +383193.697}
SPL {X  -165.650, Y  +530.452, Z    +0.000, E1   +29.664, E3 +383207.124}
SPL {X  -165.650, Y  +525.298, Z    +0.000, E1   +30.602, E3 +383218.934}
SPL {X  -165.650, Y  +518.290, Z    +0.000, E1   +31.783, E3 +383234.826}
SPL {X  -165.650, Y  +512.706, Z    +0.000, E1   +32.573, E3 +383247.661}
SPL {X  -165.650, Y  +507.785, Z    +0.000, E1   +33.438, E3 +383257.598}
SPL {X  -165.650, Y  +502.877, Z    +0.000, E1   +34.230, E3 +383267.486}
SPL {X  -165.650, Y  +499.289, Z    +0.000, E1   +34.735, E3 +383274.954}
SPL {X  -165.650, Y  +493.800, Z    +0.000, E1   +35.486, E3 +383286.326}
SPL {X  -165.650, Y  +485.583, Z    +0.000, E1   +36.670, E3 +383302.049}
SPL {X  -165.650, Y  +477.375, Z    +0.000, E1   +37.747, E3 +383317.568}
SPL {X  -165.650, Y  +469.901, Z    +0.000, E1   +38.767, E3 +383330.700}
SPL {X  -165.650, Y  +461.805, Z    +0.000, E1   +39.619, E3 +383346.043}
SPL {X  -165.650, Y  +455.681, Z    +0.000, E1   +39.641, E3 +383360.832}
SPL {X  -165.650, Y  +451.332, Z    +0.000, E1   +39.738, E3 +383370.964}
SPL {X  -165.650, Y  +448.050, Z    +0.000, E1   +39.392, E3 +383381.130}
SPL {X  -165.650, Y  +442.946, Z    +0.000, E1   +39.866, E3 +383390.905}
SPL {X  -165.650, Y  +439.091, Z    +0.000, E1   +39.674, E3 +383401.522}
SPL {X  -165.650, Y  +434.131, Z    +0.000, E1   +39.643, E3 +383414.035}
SPL {X  -165.650, Y  +428.810, Z    +0.000, E1   +39.691, E3 +383426.797}
SPL {X  -165.650, Y  +424.197, Z    +0.000, E1   +39.695, E3 +383438.156}
SPL {X  -165.650, Y  +420.220, Z    +0.000, E1   +39.526, E3 +383448.951}
SPL {X  -165.650, Y  +415.675, Z    +0.000, E1   +39.706, E3 +383459.113}
SPL {X  -165.650, Y  +410.648, Z    +0.000, E1   +39.653, E3 +383471.914}
SPL {X  -165.650, Y  +403.851, Z    +0.000, E1   +39.774, E3 +383487.999}
SPL {X  -165.650, Y  +398.253, Z    +0.000, E1   +39.688, E3 +383502.158}
SPL {X  -165.650, Y  +393.720, Z    +0.000, E1   +39.686, E3 +383513.332}
SPL {X  -165.650, Y  +389.210, Z    +0.000, E1   +39.696, E3 +383524.382}
SPL {X  -165.650, Y  +384.878, Z    +0.000, E1   +39.631, E3 +383535.458}
SPL {X  -165.650, Y  +380.529, Z    +0.000, E1   +39.528, E3 +383546.844}
SPL {X  -165.618, Y  +375.240, Z    +0.000, E1   +39.617, E3 +383559.439}
SPL {X  -165.428, Y  +369.922, Z    +0.000, E1   +39.705, E3 +383571.980}
SPL {X  -165.216, Y  +366.519, Z    +0.000, E1   +39.498, E3 +383581.547}
SPL {X  -164.790, Y  +361.646, Z    +0.000, E1   +39.684, E3 +383592.541}
SPL {X  -164.317, Y  +357.530, Z    +0.000, E1   +39.402, E3 +383604.255}
SPL {X  -163.775, Y  +353.645, Z    +0.000, E1   +39.313, E3 +383614.426}
SPL {X  -163.109, Y  +349.595, Z    +0.000, E1   +39.290, E3 +383624.487}
SPL {X  -162.309, Y  +345.398, Z    +0.000, E1   +39.085, E3 +383636.151}
SPL {X  -161.467, Y  +341.510, Z    +0.000, E1   +38.980, E3 +383646.197}
SPL {X  -160.812, Y  +338.758, Z    +0.000, E1   +38.898, E3 +383653.454}
SPL {X  -159.926, Y  +335.332, Z    +0.000, E1   +38.809, E3 +383662.411}
SPL {X  -153.020, Y  +315.059, Z    +0.000, E1   +45.580, E3 +383669.142}
SPL {X  -148.632, Y  +305.368, Z    +0.000, E1   +40.700, E3 +383728.744}
SPL {X  -145.004, Y  +298.414, Z    +0.000, E1   +40.971, E3 +383753.479}
ENDSPLINE

SPLINE
SPL {X  -149.687, Y  +307.551, Z    +0.000, E1   +36.303, E3 +383788.912}
SPL {X  -158.807, Y  +331.381, Z    +0.000, E1   +26.928, E3 +383812.564}
SPL {X  -164.505, Y  +359.058, Z    +0.000, E1   +13.887, E3 +383801.326}
SPL {X  -165.334, Y  +368.271, Z    +0.000, E1    +8.886, E3 +383799.165}
SPL {X  -165.596, Y  +374.277, Z    +0.000, E1    +5.306, E3 +383800.546}
SPL {X  -165.650, Y  +379.419, Z    +0.000, E1    +2.065, E3 +383797.568}
SPL {X  -165.650, Y  +383.176, Z    +0.000, E1    -0.610, E3 +383798.563}
SPL {X  -165.650, Y  +387.435, Z    +0.000, E1    -4.104, E3 +383796.923}
SPL {X  -165.650, Y  +393.422, Z    +0.000, E1    -9.605, E3 +383797.480}
SPL {X  -165.650, Y  +400.450, Z    +0.000, E1   -18.287, E3 +383789.295}
SPL {X  -165.650, Y  +409.248, Z    +0.000, E1   -26.478, E3 +383792.918}
SPL {X  -165.650, Y  +418.660, Z    +0.000, E1   -36.186, E3 +383790.394}
SPL {X  -165.650, Y  +444.260, Z    +0.000, E1   -47.328, E3 +383806.141}
SPL {X  -165.650, Y  +458.981, Z    +0.000, E1   -49.189, E3 +383821.685}
SPL {X  -165.650, Y  +493.049, Z    +0.000, E1   -51.657, E3 +383860.718}
ENDSPLINE

SPLINE
SPL {X  -165.650, Y  +468.984, Z    +0.000, E1   -41.461, E3 +383873.578}
SPL {X  -165.650, Y  +467.052, Z    +0.000, E1   -38.928, E3 +383884.193}
ENDSPLINE

SPLINE
SPL {X  -165.650, Y  +471.956, Z    +0.000, E1   -39.047, E3 +383895.844}
SPL {X  -165.650, Y  +478.019, Z    +0.000, E1   -39.139, E3 +383910.729}
SPL {X  -165.650, Y  +484.115, Z    +0.000, E1   -39.050, E3 +383926.490}
SPL {X  -165.650, Y  +490.374, Z    +0.000, E1   -39.169, E3 +383941.609}
SPL {X  -165.650, Y  +495.141, Z    +0.000, E1   -39.109, E3 +383953.765}
SPL {X  -165.650, Y  +497.824, Z    +0.000, E1   -38.944, E3 +383961.524}
SPL {X  -165.650, Y  +502.351, Z    +0.000, E1   -39.056, E3 +383972.407}
SPL {X  -165.650, Y  +508.180, Z    +0.000, E1   -39.157, E3 +383986.473}
SPL {X  -165.650, Y  +513.074, Z    +0.000, E1   -38.997, E3 +383999.691}
SPL {X  -165.650, Y  +518.439, Z    +0.000, E1   -39.071, E3 +384012.842}
SPL {X  -165.650, Y  +523.032, Z    +0.000, E1   -38.966, E3 +384024.978}
SPL {X  -165.650, Y  +528.401, Z    +0.000, E1   -39.135, E3 +384037.578}
SPL {X  -165.650, Y  +533.857, Z    +0.000, E1   -39.163, E3 +384051.083}
SPL {X  -165.650, Y  +539.651, Z    +0.000, E1   -39.087, E3 +384066.227}
SPL {X  -165.650, Y  +544.603, Z    +0.000, E1   -39.103, E3 +384078.403}
SPL {X  -165.650, Y  +547.280, Z    +0.000, E1   -38.965, E3 +384085.983}
SPL {X  -165.650, Y  +551.666, Z    +0.000, E1   -39.102, E3 +384096.302}
SPL {X  -165.650, Y  +555.880, Z    +0.000, E1   -39.094, E3 +384106.873}
SPL {X  -165.650, Y  +559.255, Z    +0.000, E1   -39.167, E3 +384114.909}
SPL {X  -165.650, Y  +562.850, Z    +0.000, E1   -38.959, E3 +384125.307}
SPL {X  -165.650, Y  +568.257, Z    +0.000, E1   -39.077, E3 +384138.262}
SPL {X  -165.650, Y  +573.200, Z    +0.000, E1   -39.061, E3 +384150.797}
SPL {X  -165.650, Y  +578.240, Z    +0.000, E1   -39.117, E3 +384163.138}
SPL {X  -165.650, Y  +582.804, Z    +0.000, E1   -39.080, E3 +384174.845}
SPL {X  -165.650, Y  +587.640, Z    +0.000, E1   -39.069, E3 +384187.102}
SPL {X  -165.650, Y  +592.685, Z    +0.000, E1   -39.263, E3 +384198.566}
SPL {X  -165.650, Y  +596.539, Z    +0.000, E1   -39.049, E3 +384209.555}
SPL {X  -165.650, Y  +599.973, Z    +0.000, E1   -38.814, E3 +384219.608}
SPL {X  -165.650, Y  +604.635, Z    +0.000, E1   -39.163, E3 +384229.302}
SPL {X  -165.650, Y  +608.365, Z    +0.000, E1   -39.063, E3 +384239.292}
SPL {X  -165.650, Y  +612.142, Z    +0.000, E1   -39.023, E3 +384249.022}
SPL {X  -165.650, Y  +616.635, Z    +0.000, E1   -39.260, E3 +384258.909}
SPL {X  -165.650, Y  +620.299, Z    +0.000, E1   -38.904, E3 +384270.296}
SPL {X  -165.650, Y  +625.662, Z    +0.000, E1   -39.189, E3 +384282.107}
SPL {X  -165.650, Y  +629.982, Z    +0.000, E1   -39.063, E3 +384293.708}
SPL {X  -165.650, Y  +634.317, Z    +0.000, E1   -39.239, E3 +384303.498}
SPL {X  -165.650, Y  +639.215, Z    +0.000, E1   -39.074, E3 +384317.024}
SPL {X  -165.650, Y  +643.707, Z    +0.000, E1   -38.911, E3 +384329.124}
SPL {X  -165.650, Y  +648.294, Z    +0.000, E1   -39.142, E3 +384339.379}
SPL {X  -165.650, Y  +652.477, Z    +0.000, E1   -39.068, E3 +384350.282}
SPL {X  -165.650, Y  +656.920, Z    +0.000, E1   -39.120, E3 +384361.237}
SPL {X  -165.650, Y  +662.945, Z    +0.000, E1   -39.141, E3 +384376.342}
SPL {X  -165.650, Y  +668.296, Z    +0.000, E1   -39.077, E3 +384390.067}
SPL {X  -165.650, Y  +673.138, Z    +0.000, E1   -39.196, E3 +384401.523}
SPL {X  -165.640, Y  +677.281, Z    +0.000, E1   -38.803, E3 +384414.412}
SPL {X  -165.461, Y  +683.414, Z    +0.000, E1   -39.212, E3 +384427.396}
SPL {X  -165.139, Y  +688.497, Z    +0.000, E1   -39.013, E3 +384441.448}
SPL {X  -164.582, Y  +694.282, Z    +0.000, E1   -38.975, E3 +384456.195}
SPL {X  -163.926, Y  +699.336, Z    +0.000, E1   -38.767, E3 +384470.174}
SPL {X  -163.214, Y  +703.806, Z    +0.000, E1   -38.755, E3 +384481.359}
SPL {X  -162.700, Y  +706.623, Z    +0.000, E1   -38.580, E3 +384489.471}
SPL {X  -161.983, Y  +710.160, Z    +0.000, E1   -38.439, E3 +384499.251}
SPL {X  -161.163, Y  +713.794, Z    +0.000, E1   -38.390, E3 +384508.621}
SPL {X  -160.158, Y  +717.801, Z    +0.000, E1   -38.225, E3 +384519.751}
SPL {X  -155.870, Y  +731.575, Z    +0.000, E1   -42.661, E3 +384527.214}
SPL {X  -137.799, Y  +767.431, Z    +0.000, E1   -46.550, E3 +384583.724}
ENDSPLINE

SPLINE
SPL {X  -141.948, Y  +760.885, Z    +0.000, E1   -42.258, E3 +384615.860}
SPL {X  -160.264, Y  +717.397, Z    +0.000, E1   -24.835, E3 +384657.044}
SPL {X  -164.762, Y  +692.628, Z    +0.000, E1   -12.660, E3 +384660.297}
SPL {X  -165.481, Y  +682.990, Z    +0.000, E1    -7.255, E3 +384657.141}
SPL {X  -165.649, Y  +676.021, Z    +0.000, E1    -3.061, E3 +384654.509}
SPL {X  -165.650, Y  +670.589, Z    +0.000, E1    +0.778, E3 +384653.746}
SPL {X  -165.650, Y  +666.842, Z    +0.000, E1    +3.871, E3 +384653.207}
SPL {X  -165.650, Y  +662.773, Z    +0.000, E1    +7.549, E3 +384653.352}
SPL {X  -165.650, Y  +656.581, Z    +0.000, E1   +13.870, E3 +384651.402}
SPL {X  -165.650, Y  +648.120, Z    +0.000, E1   +22.794, E3 +384650.633}
SPL {X  -165.650, Y  +632.103, Z    +0.000, E1   +42.949, E3 +384637.591}
SPL {X  -165.650, Y  +608.448, Z    +0.000, E1   +47.265, E3 +384664.031}
SPL {X  -165.650, Y  +595.526, Z    +0.000, E1   +48.856, E3 +384677.889}
SPL {X  -165.650, Y  +568.828, Z    +0.000, E1   +48.639, E3 +384720.442}
ENDSPLINE

SPLINE
SPL {X  -165.650, Y  +587.144, Z    +0.000, E1   +39.840, E3 +384734.474}
ENDSPLINE

SPLINE
SPL {X  -165.650, Y  +582.480, Z    +0.000, E1   +38.929, E3 +384751.670}
SPL {X  -165.650, Y  +576.923, Z    +0.000, E1   +38.908, E3 +384765.700}
SPL {X  -165.650, Y  +571.957, Z    +0.000, E1   +38.951, E3 +384778.105}
SPL {X  -165.650, Y  +566.463, Z    +0.000, E1   +38.933, E3 +384792.077}
SPL {X  -165.650, Y  +561.565, Z    +0.000, E1   +38.903, E3 +384804.651}
SPL {X  -165.650, Y  +555.731, Z    +0.000, E1   +38.913, E3 +384819.508}
SPL {X  -165.650, Y  +549.409, Z    +0.000, E1   +38.884, E3 +384835.657}
SPL {X  -165.650, Y  +544.480, Z    +0.000, E1   +38.998, E3 +384847.320}
SPL {X  -165.650, Y  +540.151, Z    +0.000, E1   +38.996, E3 +384858.366}
SPL {X  -165.650, Y  +534.008, Z    +0.000, E1   +38.962, E3 +384874.208}
SPL {X  -165.650, Y  +528.320, Z    +0.000, E1   +38.809, E3 +384889.445}
SPL {X  -165.650, Y  +524.195, Z    +0.000, E1   +38.844, E3 +384899.621}
SPL {X  -165.650, Y  +520.666, Z    +0.000, E1   +39.043, E3 +384907.346}
ENDSPLINE

SPLINE
SPL {X  -165.650, Y  +541.168, Z    +0.000, E1   +27.957, E3 +384915.904}
ENDSPLINE

SPLINE
SPL {X  -165.650, Y  +536.052, Z    +0.000, E1   +28.653, E3 +384930.539}
SPL {X  -165.650, Y  +530.452, Z    +0.000, E1   +29.664, E3 +384943.966}
SPL {X  -165.650, Y  +523.712, Z    +0.000, E1   +30.911, E3 +384959.248}
SPL {X  -165.650, Y  +516.975, Z    +0.000, E1   +31.942, E3 +384974.842}
SPL {X  -165.650, Y  +512.706, Z    +0.000, E1   +32.573, E3 +384984.503}
SPL {X  -165.650, Y  +507.785, Z    +0.000, E1   +33.438, E3 +384994.440}
SPL {X  -165.650, Y  +501.257, Z    +0.000, E1   +34.478, E3 +385007.680}
SPL {X  -165.650, Y  +495.236, Z    +0.000, E1   +35.288, E3 +385020.185}
SPL {X  -165.650, Y  +488.684, Z    +0.000, E1   +36.217, E3 +385033.082}
SPL {X  -165.650, Y  +483.157, Z    +0.000, E1   +36.957, E3 +385043.645}
SPL {X  -165.650, Y  +477.375, Z    +0.000, E1   +37.747, E3 +385054.410}
SPL {X  -165.650, Y  +469.901, Z    +0.000, E1   +38.767, E3 +385067.542}
SPL {X  -165.650, Y  +461.805, Z    +0.000, E1   +39.619, E3 +385082.885}
SPL {X  -165.650, Y  +455.681, Z    +0.000, E1   +39.641, E3 +385097.674}
SPL {X  -165.650, Y  +451.332, Z    +0.000, E1   +39.738, E3 +385107.806}
SPL {X  -165.650, Y  +448.050, Z    +0.000, E1   +39.392, E3 +385117.972}
SPL {X  -165.650, Y  +442.946, Z    +0.000, E1   +39.866, E3 +385127.747}
SPL {X  -165.650, Y  +439.091, Z    +0.000, E1   +39.674, E3 +385138.365}
SPL {X  -165.650, Y  +434.131, Z    +0.000, E1   +39.643, E3 +385150.877}
SPL {X  -165.650, Y  +428.810, Z    +0.000, E1   +39.691, E3 +385163.639}
SPL {X  -165.650, Y  +424.197, Z    +0.000, E1   +39.695, E3 +385174.998}
SPL {X  -165.650, Y  +420.220, Z    +0.000, E1   +39.526, E3 +385185.793}
SPL {X  -165.650, Y  +414.177, Z    +0.000, E1   +39.693, E3 +385199.920}
SPL {X  -165.650, Y  +407.394, Z    +0.000, E1   +39.797, E3 +385215.875}
SPL {X  -165.650, Y  +402.798, Z    +0.000, E1   +39.651, E3 +385227.996}
SPL {X  -165.650, Y  +398.253, Z    +0.000, E1   +39.688, E3 +385239.000}
SPL {X  -165.650, Y  +393.720, Z    +0.000, E1   +39.686, E3 +385250.174}
SPL {X  -165.650, Y  +389.210, Z    +0.000, E1   +39.696, E3 +385261.224}
SPL {X  -165.650, Y  +384.878, Z    +0.000, E1   +39.631, E3 +385272.300}
SPL {X  -165.650, Y  +380.529, Z    +0.000, E1   +39.528, E3 +385283.687}
SPL {X  -165.618, Y  +375.240, Z    +0.000, E1   +39.617, E3 +385296.281}
SPL {X  -165.428, Y  +369.922, Z    +0.000, E1   +39.705, E3 +385308.822}
SPL {X  -165.216, Y  +366.519, Z    +0.000, E1   +39.498, E3 +385318.389}
SPL {X  -164.790, Y  +361.646, Z    +0.000, E1   +39.684, E3 +385329.384}
SPL {X  -164.317, Y  +357.530, Z    +0.000, E1   +39.402, E3 +385341.097}
SPL {X  -163.775, Y  +353.645, Z    +0.000, E1   +39.313, E3 +385351.268}
SPL {X  -163.109, Y  +349.595, Z    +0.000, E1   +39.290, E3 +385361.329}
SPL {X  -162.309, Y  +345.398, Z    +0.000, E1   +39.085, E3 +385372.993}
SPL {X  -161.467, Y  +341.510, Z    +0.000, E1   +38.980, E3 +385383.039}
SPL {X  -160.812, Y  +338.758, Z    +0.000, E1   +38.898, E3 +385390.296}
SPL {X  -159.926, Y  +335.332, Z    +0.000, E1   +38.809, E3 +385399.253}
SPL {X  -153.020, Y  +315.059, Z    +0.000, E1   +45.580, E3 +385405.984}
SPL {X  -148.632, Y  +305.368, Z    +0.000, E1   +40.700, E3 +385465.586}
SPL {X  -145.004, Y  +298.414, Z    +0.000, E1   +40.971, E3 +385490.322}
ENDSPLINE

SPLINE
SPL {X  -149.687, Y  +307.551, Z    +0.000, E1   +36.303, E3 +385525.754}
SPL {X  -158.807, Y  +331.381, Z    +0.000, E1   +26.928, E3 +385549.406}
SPL {X  -164.505, Y  +359.058, Z    +0.000, E1   +13.887, E3 +385538.168}
SPL {X  -165.494, Y  +371.321, Z    +0.000, E1    +7.176, E3 +385536.729}
SPL {X  -165.650, Y  +379.419, Z    +0.000, E1    +2.065, E3 +385534.410}
SPL {X  -165.650, Y  +383.176, Z    +0.000, E1    -0.610, E3 +385535.405}
SPL {X  -165.650, Y  +387.435, Z    +0.000, E1    -4.104, E3 +385533.765}
SPL {X  -165.650, Y  +393.422, Z    +0.000, E1    -9.605, E3 +385534.322}
SPL {X  -165.650, Y  +400.450, Z    +0.000, E1   -18.287, E3 +385526.137}
SPL {X  -165.650, Y  +409.248, Z    +0.000, E1   -26.478, E3 +385529.760}
SPL {X  -165.650, Y  +418.660, Z    +0.000, E1   -36.186, E3 +385527.236}
SPL {X  -165.650, Y  +444.260, Z    +0.000, E1   -47.328, E3 +385542.984}
SPL {X  -165.650, Y  +458.981, Z    +0.000, E1   -49.189, E3 +385558.527}
SPL {X  -165.650, Y  +493.049, Z    +0.000, E1   -51.657, E3 +385597.560}
ENDSPLINE

SPLINE
SPL {X  -165.650, Y  +468.984, Z    +0.000, E1   -41.461, E3 +385610.420}
SPL {X  -165.650, Y  +467.052, Z    +0.000, E1   -38.928, E3 +385621.035}
ENDSPLINE

